LIN {X 0,Y 331.021,Z 915.228,A -85,B 0,C 180,E1 16163.029,E2 16163.029} C_VEL
LIN {X 0,Y 337.133,Z 895.779,A -85,B 0,C 180,E1 16164.723,E2 16164.723} C_VEL
LIN {X 0,Y 338.679,Z 881.099,A -85,B 0,C 180,E1 16166.333,E2 16166.333} C_VEL
LIN {X 0,Y 339.674,Z 868.031,A -85,B 0,C 180,E1 16167.682,E2 16167.682} C_VEL
LIN {X 0,Y 340.17,Z 866.046,A -85,B 0,C 180,E1 16167.812,E2 16167.812} C_VEL
LIN {X 0,Y 341.218,Z 861.378,A -85,B 0,C 180,E1 16168.096,E2 16168.096} C_VEL
LIN {X 0,Y 333.256,Z 836.302,A -85,B 0,C 180,E1 16172.609,E2 16172.609} C_VEL
LIN {X 0,Y 322.714,Z 812.784,A -85,B 0,C 180,E1 16178.041,E2 16178.041} C_VEL
LIN {X 0,Y 312.358,Z 794.085,A -85,B 0,C 180,E1 16183.992,E2 16183.992} C_VEL
LIN {X 0,Y 304.44,Z 781.718,A -85,B 0,C 180,E1 16189.789,E2 16189.789} C_VEL
LIN {X 0,Y 300.25,Z 775.211,A -85,B 0,C 180,E1 16194.023,E2 16194.023} C_VEL
LIN {X 0,Y 297.058,Z 768.999,A -85,B 0,C 180,E1 16199.536,E2 16199.536} C_VEL
LIN {X 0,Y 296.553,Z 769.306,A -85,B 0,C 180,E1 16209.301,E2 16209.301} C_VEL
LIN {X 0,Y 299.386,Z 775.096,A -85,B 0,C 180,E1 16215.012,E2 16215.012} C_VEL
LIN {X 0,Y 301.02,Z 777.25,A -85,B 0,C 180,E1 16217.046,E2 16217.046} C_VEL
LIN {X 0,Y 305.693,Z 785.45,A -85,B 0,C 180,E1 16221.795,E2 16221.795} C_VEL
LIN {X 0,Y 311.815,Z 796.017,A -85,B 0,C 180,E1 16226.634,E2 16226.634} C_VEL
LIN {X 0,Y 320.081,Z 813.536,A -85,B 0,C 180,E1 16232.477,E2 16232.477} C_VEL
LIN {X 0,Y 327.738,Z 835.588,A -85,B 0,C 180,E1 16238.25,E2 16238.25} C_VEL
LIN {X 0,Y 332.514,Z 859.666,A -85,B 0,C 180,E1 16243.601,E2 16243.601} C_VEL
LIN {X 0,Y 330.699,Z 866.985,A -85,B 0,C 180,E1 16244.544,E2 16244.544} C_VEL
LIN {X 0,Y 318.48,Z 897.247,A -85,B 0,C 180,E1 16248.528,E2 16248.528} C_VEL
LIN {X 0,Y 305.736,Z 923.66,A -85,B 0,C 180,E1 16253.542,E2 16253.542} C_VEL
LIN {X 0,Y 294.077,Z 945.097,A -85,B 0,C 180,E1 16259.443,E2 16259.443} C_VEL
LIN {X 0,Y 284.318,Z 962.198,A -85,B 0,C 180,E1 16266.461,E2 16266.461} C_VEL
LIN {X 0,Y 277.725,Z 974.062,A -85,B 0,C 180,E1 16274.183,E2 16274.183} C_VEL
LIN {X 0,Y 274.803,Z 979.693,A -85,B 0,C 180,E1 16280.487,E2 16280.487} C_VEL
LIN {X 0,Y 273.739,Z 982.416,A -85,B 0,C 180,E1 16286.83,E2 16286.83} C_VEL
LIN {X 0,Y 273.747,Z 982.384,A -85,B 0,C 180,E1 16293.171,E2 16293.171} C_VEL
LIN {X 0,Y 275.395,Z 978.493,A -85,B 0,C 180,E1 16301.094,E2 16301.094} C_VEL
LIN {X 0,Y 279.926,Z 969.8,A -85,B 0,C 180,E1 16308.936,E2 16308.936} C_VEL
LIN {X 0,Y 287.816,Z 955.85,A -85,B 0,C 180,E1 16316.395,E2 16316.395} C_VEL
LIN {X 0,Y 298.558,Z 936.897,A -85,B 0,C 180,E1 16322.978,E2 16322.978} C_VEL
LIN {X 0,Y 310.721,Z 913.541,A -85,B 0,C 180,E1 16328.506,E2 16328.506} C_VEL
LIN {X 0,Y 323.773,Z 884.724,A -85,B 0,C 180,E1 16333.206,E2 16333.206} C_VEL
LIN {X 0,Y 332.594,Z 860.778,A -85,B 0,C 180,E1 16336.051,E2 16336.051} C_VEL
LIN {X 0,Y 327.799,Z 836.283,A -85,B 0,C 180,E1 16341.479,E2 16341.479} C_VEL
LIN {X 0,Y 320.691,Z 815.062,A -85,B 0,C 180,E1 16346.924,E2 16346.924} C_VEL
LIN {X 0,Y 311.788,Z 796.082,A -85,B 0,C 180,E1 16353.185,E2 16353.185} C_VEL
LIN {X 0,Y 304.22,Z 782.321,A -85,B 0,C 180,E1 16359.432,E2 16359.432} C_VEL
LIN {X 0,Y 300.038,Z 775.489,A -85,B 0,C 180,E1 16363.895,E2 16363.895} C_VEL
LIN {X 0,Y 296.56,Z 769.453,A -85,B 0,C 180,E1 16369.925,E2 16369.925} C_VEL
LIN {X 0,Y 296.669,Z 768.461,A -85,B 0,C 180,E1 16380.008,E2 16380.008} C_VEL
LIN {X 0,Y 300.732,Z 775.566,A -85,B 0,C 180,E1 16386.693,E2 16386.693} C_VEL
LIN {X 0,Y 306.504,Z 785.112,A -85,B 0,C 180,E1 16392.034,E2 16392.034} C_VEL
LIN {X 0,Y 313.542,Z 796.189,A -85,B 0,C 180,E1 16396.847,E2 16396.847} C_VEL
LIN {X 0,Y 324.459,Z 816.254,A -85,B 0,C 180,E1 16402.919,E2 16402.919} C_VEL
LIN {X 0,Y 334.954,Z 840.847,A -85,B 0,C 180,E1 16408.338,E2 16408.338} C_VEL
LIN {X 0,Y 341.11,Z 861.37,A -85,B 0,C 180,E1 16411.908,E2 16411.908} C_VEL
LIN {X 0,Y 329.462,Z 902.909,A -85,B 0,C 180,E1 16414.862,E2 16414.862} C_VEL
LIN {X 0,Y 315.546,Z 942.717,A -85,B 0,C 180,E1 16419.055,E2 16419.055} C_VEL
LIN {X 0,Y 302.271,Z 976.846,A -85,B 0,C 180,E1 16424.232,E2 16424.232} C_VEL
LIN {X 0,Y 290.023,Z 1007.512,A -85,B 0,C 180,E1 16430.731,E2 16430.731} C_VEL
LIN {X 0,Y 280.658,Z 1033.018,A -85,B 0,C 180,E1 16438.227,E2 16438.227} C_VEL
LIN {X 0,Y 274.674,Z 1053.485,A -85,B 0,C 180,E1 16446.65,E2 16446.65} C_VEL
LIN {X 0,Y 272.304,Z 1067.457,A -85,B 0,C 180,E1 16455.096,E2 16455.096} C_VEL
LIN {X 0,Y 271.923,Z 1074.33,A -85,B 0,C 180,E1 16461.999,E2 16461.999} C_VEL
LIN {X 0,Y 272.108,Z 1076.824,A -85,B 0,C 180,E1 16466.81,E2 16466.81} C_VEL
LIN {X 0,Y 272.364,Z 1077.339,A -85,B 0,C 180,E1 16470,E2 16470} C_VEL
LIN {X 0,Y 272.002,Z 1075.42,A -85,B 0,C 180,E1 16476.391,E2 16476.391} C_VEL
LIN {X 0,Y 272.256,Z 1067.956,A -85,B 0,C 180,E1 16484.492,E2 16484.492} C_VEL
LIN {X 0,Y 274.36,Z 1054.719,A -85,B 0,C 180,E1 16492.723,E2 16492.723} C_VEL
LIN {X 0,Y 279.536,Z 1036.37,A -85,B 0,C 180,E1 16500.582,E2 16500.582} C_VEL
LIN {X 0,Y 288.648,Z 1011.145,A -85,B 0,C 180,E1 16508.341,E2 16508.341} C_VEL
LIN {X 0,Y 300.414,Z 981.675,A -85,B 0,C 180,E1 16514.874,E2 16514.874} C_VEL
LIN {X 0,Y 313.155,Z 949.302,A -85,B 0,C 180,E1 16520.072,E2 16520.072} C_VEL
LIN {X 0,Y 326.1,Z 913.314,A -85,B 0,C 180,E1 16524.199,E2 16524.199} C_VEL
LIN {X 0,Y 338.026,Z 873.973,A -85,B 0,C 180,E1 16527.32,E2 16527.32} C_VEL
LIN {X 0,Y 340.17,Z 866.046,A -85,B 0,C 180,E1 16527.812,E2 16527.812} C_VEL
LIN {X 0,Y 339.446,Z 860.887,A -85,B 0,C 180,E1 16528.559,E2 16528.559} C_VEL
LIN {X 0,Y 332.595,Z 853.241,A -85,B 0,C 180,E1 16530.955,E2 16530.955} C_VEL
LIN {X 0,Y 323.201,Z 827.838,A -85,B 0,C 180,E1 16536.348,E2 16536.348} C_VEL
LIN {X 0,Y 313.242,Z 807.134,A -85,B 0,C 180,E1 16542.23,E2 16542.23} C_VEL
LIN {X 0,Y 305.313,Z 793.908,A -85,B 0,C 180,E1 16547.736,E2 16547.736} C_VEL
LIN {X 0,Y 301.561,Z 787.929,A -85,B 0,C 180,E1 16551.058,E2 16551.058} C_VEL
LIN {X 0,Y 298.756,Z 782.824,A -85,B 0,C 180,E1 16554.358,E2 16554.358} C_VEL
LIN {X 0,Y 295.744,Z 776.422,A -85,B 0,C 180,E1 16559.992,E2 16559.992} C_VEL
LIN {X 0,Y 295.279,Z 777.204,A -85,B 0,C 180,E1 16569.164,E2 16569.164} C_VEL
LIN {X 0,Y 298.129,Z 783.012,A -85,B 0,C 180,E1 16575.301,E2 16575.301} C_VEL
LIN {X 0,Y 302.957,Z 791.913,A -85,B 0,C 180,E1 16581.04,E2 16581.04} C_VEL
LIN {X 0,Y 308.902,Z 803.163,A -85,B 0,C 180,E1 16586.27,E2 16586.27} C_VEL
LIN {X 0,Y 316.328,Z 820.365,A -85,B 0,C 180,E1 16592.16,E2 16592.16} C_VEL
LIN {X 0,Y 322.984,Z 841.616,A -85,B 0,C 180,E1 16597.876,E2 16597.876} C_VEL
LIN {X 0,Y 326.886,Z 864.273,A -85,B 0,C 180,E1 16603.076,E2 16603.076} C_VEL
LIN {X 0,Y 314.014,Z 895.921,A -85,B 0,C 180,E1 16607.129,E2 16607.129} C_VEL
LIN {X 0,Y 300.859,Z 922.582,A -85,B 0,C 180,E1 16612.083,E2 16612.083} C_VEL
LIN {X 0,Y 289.103,Z 943.576,A -85,B 0,C 180,E1 16617.687,E2 16617.687} C_VEL
LIN {X 0,Y 278.977,Z 960.478,A -85,B 0,C 180,E1 16624.269,E2 16624.269} C_VEL
LIN {X 0,Y 271.013,Z 973.81,A -85,B 0,C 180,E1 16632.406,E2 16632.406} C_VEL
LIN {X 0,Y 267.113,Z 981.045,A -85,B 0,C 180,E1 16640.21,E2 16640.21} C_VEL
LIN {X 0,Y 265.969,Z 983.764,A -85,B 0,C 180,E1 16646.737,E2 16646.737} C_VEL
LIN {X 0,Y 265.977,Z 983.732,A -85,B 0,C 180,E1 16653.263,E2 16653.263} C_VEL
LIN {X 0,Y 267.761,Z 979.844,A -85,B 0,C 180,E1 16661.414,E2 16661.414} C_VEL
LIN {X 0,Y 272.543,Z 971.167,A -85,B 0,C 180,E1 16669.47,E2 16669.47} C_VEL
LIN {X 0,Y 280.895,Z 957.141,A -85,B 0,C 180,E1 16677.143,E2 16677.143} C_VEL
LIN {X 0,Y 291.909,Z 938.548,A -85,B 0,C 180,E1 16683.739,E2 16683.739} C_VEL
LIN {X 0,Y 304.564,Z 915.214,A -85,B 0,C 180,E1 16689.374,E2 16689.374} C_VEL
LIN {X 0,Y 317.442,Z 887.919,A -85,B 0,C 180,E1 16693.931,E2 16693.931} C_VEL
LIN {X 0,Y 326.74,Z 863.857,A -85,B 0,C 180,E1 16696.906,E2 16696.906} C_VEL
LIN {X 0,Y 322.479,Z 840.057,A -85,B 0,C 180,E1 16702.399,E2 16702.399} C_VEL
LIN {X 0,Y 316.105,Z 820.038,A -85,B 0,C 180,E1 16707.814,E2 16707.814} C_VEL
LIN {X 0,Y 308.12,Z 801.577,A -85,B 0,C 180,E1 16714.168,E2 16714.168} C_VEL
LIN {X 0,Y 301.32,Z 789.044,A -85,B 0,C 180,E1 16720.375,E2 16720.375} C_VEL
LIN {X 0,Y 297.981,Z 782.896,A -85,B 0,C 180,E1 16724.538,E2 16724.538} C_VEL
LIN {X 0,Y 295.21,Z 776.702,A -85,B 0,C 180,E1 16730.495,E2 16730.495} C_VEL
LIN {X 0,Y 295.719,Z 776.954,A -85,B 0,C 180,E1 16740.649,E2 16740.649} C_VEL
LIN {X 0,Y 299.033,Z 783.061,A -85,B 0,C 180,E1 16746.183,E2 16746.183} C_VEL
LIN {X 0,Y 304.41,Z 792.508,A -85,B 0,C 180,E1 16751.663,E2 16751.663} C_VEL
LIN {X 0,Y 311.029,Z 803.407,A -85,B 0,C 180,E1 16756.442,E2 16756.442} C_VEL
LIN {X 0,Y 320.973,Z 822.87,A -85,B 0,C 180,E1 16762.449,E2 16762.449} C_VEL
LIN {X 0,Y 330.869,Z 847.763,A -85,B 0,C 180,E1 16768.028,E2 16768.028} C_VEL
LIN {X 0,Y 335.299,Z 865.581,A -85,B 0,C 180,E1 16771.117,E2 16771.117} C_VEL
LIN {X 0,Y 323.255,Z 905.592,A -85,B 0,C 180,E1 16774.067,E2 16774.067} C_VEL
LIN {X 0,Y 309.246,Z 943.627,A -85,B 0,C 180,E1 16778.197,E2 16778.197} C_VEL
LIN {X 0,Y 295.249,Z 977.945,A -85,B 0,C 180,E1 16783.568,E2 16783.568} C_VEL
LIN {X 0,Y 282.871,Z 1007.45,A -85,B 0,C 180,E1 16790.039,E2 16790.039} C_VEL
LIN {X 0,Y 273.077,Z 1032.74,A -85,B 0,C 180,E1 16797.749,E2 16797.749} C_VEL
LIN {X 0,Y 267.231,Z 1051.564,A -85,B 0,C 180,E1 16805.703,E2 16805.703} C_VEL
LIN {X 0,Y 264.59,Z 1065.504,A -85,B 0,C 180,E1 16814.229,E2 16814.229} C_VEL
LIN {X 0,Y 264.096,Z 1072.957,A -85,B 0,C 180,E1 16821.76,E2 16821.76} C_VEL
LIN {X 0,Y 264.307,Z 1075.47,A -85,B 0,C 180,E1 16826.716,E2 16826.716} C_VEL
LIN {X 0,Y 264.598,Z 1075.994,A -85,B 0,C 180,E1 16830,E2 16830} C_VEL
LIN {X 0,Y 264.197,Z 1074.056,A -85,B 0,C 180,E1 16836.581,E2 16836.581} C_VEL
LIN {X 0,Y 264.316,Z 1068.494,A -85,B 0,C 180,E1 16843.245,E2 16843.245} C_VEL
LIN {X 0,Y 266.059,Z 1056.461,A -85,B 0,C 180,E1 16851.708,E2 16851.708} C_VEL
LIN {X 0,Y 271.419,Z 1037.536,A -85,B 0,C 180,E1 16860.495,E2 16860.495} C_VEL
LIN {X 0,Y 280.433,Z 1013.604,A -85,B 0,C 180,E1 16868.343,E2 16868.343} C_VEL
LIN {X 0,Y 292.855,Z 983.925,A -85,B 0,C 180,E1 16875.303,E2 16875.303} C_VEL
LIN {X 0,Y 306.741,Z 950.365,A -85,B 0,C 180,E1 16880.896,E2 16880.896} C_VEL
LIN {X 0,Y 320.69,Z 913.175,A -85,B 0,C 180,E1 16885.243,E2 16885.243} C_VEL
LIN {X 0,Y 332.946,Z 874.288,A -85,B 0,C 180,E1 16888.358,E2 16888.358} C_VEL
LIN {X 0,Y 335.623,Z 864.362,A -85,B 0,C 180,E1 16888.991,E2 16888.991} C_VEL
LIN {X 0,Y 332.595,Z 853.241,A -85,B 0,C 180,E1 16890.955,E2 16890.955} C_VEL
LIN {X 0,Y 328.462,Z 846.564,A -85,B 0,C 180,E1 16892.778,E2 16892.778} C_VEL
LIN {X 0,Y 320.655,Z 837.361,A -85,B 0,C 180,E1 16896.065,E2 16896.065} C_VEL
LIN {X 0,Y 311.653,Z 817.013,A -85,B 0,C 180,E1 16901.77,E2 16901.77} C_VEL
LIN {X 0,Y 304.174,Z 802.822,A -85,B 0,C 180,E1 16907.233,E2 16907.233} C_VEL
LIN {X 0,Y 299.303,Z 794.888,A -85,B 0,C 180,E1 16911.722,E2 16911.722} C_VEL
LIN {X 0,Y 296.792,Z 790.23,A -85,B 0,C 180,E1 16914.871,E2 16914.871} C_VEL
LIN {X 0,Y 294.14,Z 784.145,A -85,B 0,C 180,E1 16920.61,E2 16920.61} C_VEL
LIN {X 0,Y 293.722,Z 784.97,A -85,B 0,C 180,E1 16928.968,E2 16928.968} C_VEL
LIN {X 0,Y 296.55,Z 790.82,A -85,B 0,C 180,E1 16935.482,E2 16935.482} C_VEL
LIN {X 0,Y 301.16,Z 800.76,A -85,B 0,C 180,E1 16941.462,E2 16941.462} C_VEL
LIN {X 0,Y 306.312,Z 811.538,A -85,B 0,C 180,E1 16946.402,E2 16946.402} C_VEL
LIN {X 0,Y 312.882,Z 828.141,A -85,B 0,C 180,E1 16952.148,E2 16952.148} C_VEL
LIN {X 0,Y 318.462,Z 848.77,A -85,B 0,C 180,E1 16957.799,E2 16957.799} C_VEL
LIN {X 0,Y 320.811,Z 868.378,A -85,B 0,C 180,E1 16962.364,E2 16962.364} C_VEL
LIN {X 0,Y 308.216,Z 897.773,A -85,B 0,C 180,E1 16966.206,E2 16966.206} C_VEL
LIN {X 0,Y 294.886,Z 923.817,A -85,B 0,C 180,E1 16971.112,E2 16971.112} C_VEL
LIN {X 0,Y 282.334,Z 945.309,A -85,B 0,C 180,E1 16976.958,E2 16976.958} C_VEL
LIN {X 0,Y 271.966,Z 961.846,A -85,B 0,C 180,E1 16983.555,E2 16983.555} C_VEL
LIN {X 0,Y 264.131,Z 974.24,A -85,B 0,C 180,E1 16991.125,E2 16991.125} C_VEL
LIN {X 0,Y 259.45,Z 982.392,A -85,B 0,C 180,E1 16999.918,E2 16999.918} C_VEL
LIN {X 0,Y 258.208,Z 985.111,A -85,B 0,C 180,E1 17006.639,E2 17006.639} C_VEL
LIN {X 0,Y 258.217,Z 985.079,A -85,B 0,C 180,E1 17013.362,E2 17013.362} C_VEL
LIN {X 0,Y 260.137,Z 981.196,A -85,B 0,C 180,E1 17021.754,E2 17021.754} C_VEL
LIN {X 0,Y 265.186,Z 972.532,A -85,B 0,C 180,E1 17030.033,E2 17030.033} C_VEL
LIN {X 0,Y 273.959,Z 958.549,A -85,B 0,C 180,E1 17037.872,E2 17037.872} C_VEL
LIN {X 0,Y 285.458,Z 939.958,A -85,B 0,C 180,E1 17044.608,E2 17044.608} C_VEL
LIN {X 0,Y 298.643,Z 916.602,A -85,B 0,C 180,E1 17050.333,E2 17050.333} C_VEL
LIN {X 0,Y 312.136,Z 888.985,A -85,B 0,C 180,E1 17054.985,E2 17054.985} C_VEL
LIN {X 0,Y 320.922,Z 866.987,A -85,B 0,C 180,E1 17057.772,E2 17057.772} C_VEL
LIN {X 0,Y 317.398,Z 844.495,A -85,B 0,C 180,E1 17063.182,E2 17063.182} C_VEL
LIN {X 0,Y 311.442,Z 824.288,A -85,B 0,C 180,E1 17068.913,E2 17068.913} C_VEL
LIN {X 0,Y 304.534,Z 807.578,A -85,B 0,C 180,E1 17075.06,E2 17075.06} C_VEL
LIN {X 0,Y 298.817,Z 796.122,A -85,B 0,C 180,E1 17080.974,E2 17080.974} C_VEL
LIN {X 0,Y 296.046,Z 790.466,A -85,B 0,C 180,E1 17084.815,E2 17084.815} C_VEL
LIN {X 0,Y 293.489,Z 784.102,A -85,B 0,C 180,E1 17091.354,E2 17091.354} C_VEL
LIN {X 0,Y 294.251,Z 784.854,A -85,B 0,C 180,E1 17100.484,E2 17100.484} C_VEL
LIN {X 0,Y 298.156,Z 792.625,A -85,B 0,C 180,E1 17107.117,E2 17107.117} C_VEL
LIN {X 0,Y 303.043,Z 801.272,A -85,B 0,C 180,E1 17111.991,E2 17111.991} C_VEL
LIN {X 0,Y 310.547,Z 814.766,A -85,B 0,C 180,E1 17117.563,E2 17117.563} C_VEL
LIN {X 0,Y 319.314,Z 834.216,A -85,B 0,C 180,E1 17123.176,E2 17123.176} C_VEL
LIN {X 0,Y 327.303,Z 857.161,A -85,B 0,C 180,E1 17128.233,E2 17128.233} C_VEL
LIN {X 0,Y 329.873,Z 867.279,A -85,B 0,C 180,E1 17130.105,E2 17130.105} C_VEL
LIN {X 0,Y 317.632,Z 906.603,A -85,B 0,C 180,E1 17133.096,E2 17133.096} C_VEL
LIN {X 0,Y 303.691,Z 942.962,A -85,B 0,C 180,E1 17137.094,E2 17137.094} C_VEL
LIN {X 0,Y 289.455,Z 976.399,A -85,B 0,C 180,E1 17142.37,E2 17142.37} C_VEL
LIN {X 0,Y 276.484,Z 1005.907,A -85,B 0,C 180,E1 17148.92,E2 17148.92} C_VEL
LIN {X 0,Y 265.97,Z 1031.227,A -85,B 0,C 180,E1 17156.778,E2 17156.778} C_VEL
LIN {X 0,Y 259.706,Z 1050.107,A -85,B 0,C 180,E1 17164.951,E2 17164.951} C_VEL
LIN {X 0,Y 256.828,Z 1064.091,A -85,B 0,C 180,E1 17173.739,E2 17173.739} C_VEL
LIN {X 0,Y 256.281,Z 1071.587,A -85,B 0,C 180,E1 17181.507,E2 17181.507} C_VEL
LIN {X 0,Y 256.513,Z 1074.116,A -85,B 0,C 180,E1 17186.616,E2 17186.616} C_VEL
LIN {X 0,Y 256.824,Z 1074.647,A -85,B 0,C 180,E1 17190,E2 17190} C_VEL
LIN {X 0,Y 256.363,Z 1072.688,A -85,B 0,C 180,E1 17196.783,E2 17196.783} C_VEL
LIN {X 0,Y 256.514,Z 1067.096,A -85,B 0,C 180,E1 17203.655,E2 17203.655} C_VEL
LIN {X 0,Y 258.399,Z 1055.007,A -85,B 0,C 180,E1 17212.386,E2 17212.386} C_VEL
LIN {X 0,Y 264.325,Z 1035.788,A -85,B 0,C 180,E1 17221.51,E2 17221.51} C_VEL
LIN {X 0,Y 274.32,Z 1010.866,A -85,B 0,C 180,E1 17229.767,E2 17229.767} C_VEL
LIN {X 0,Y 287.754,Z 980.553,A -85,B 0,C 180,E1 17236.838,E2 17236.838} C_VEL
LIN {X 0,Y 301.735,Z 948.101,A -85,B 0,C 180,E1 17242.211,E2 17242.211} C_VEL
LIN {X 0,Y 315.862,Z 911.832,A -85,B 0,C 180,E1 17246.427,E2 17246.427} C_VEL
LIN {X 0,Y 328.463,Z 872.948,A -85,B 0,C 180,E1 17249.529,E2 17249.529} C_VEL
LIN {X 0,Y 329.734,Z 866.231,A -85,B 0,C 180,E1 17250.095,E2 17250.095} C_VEL
LIN {X 0,Y 322.374,Z 841.982,A -85,B 0,C 180,E1 17254.991,E2 17254.991} C_VEL
LIN {X 0,Y 320.655,Z 837.361,A -85,B 0,C 180,E1 17256.065,E2 17256.065} C_VEL
LIN {X 0,Y 315.045,Z 830.532,A -85,B 0,C 180,E1 17258.785,E2 17258.785} C_VEL
LIN {X 0,Y 309.157,Z 825.25,A -85,B 0,C 180,E1 17261.716,E2 17261.716} C_VEL
LIN {X 0,Y 301.715,Z 810.065,A -85,B 0,C 180,E1 17267.588,E2 17267.588} C_VEL
LIN {X 0,Y 295.456,Z 798.281,A -85,B 0,C 180,E1 17274.486,E2 17274.486} C_VEL
LIN {X 0,Y 292.411,Z 791.833,A -85,B 0,C 180,E1 17281.236,E2 17281.236} C_VEL
LIN {X 0,Y 292.006,Z 792.598,A -85,B 0,C 180,E1 17288.705,E2 17288.705} C_VEL
LIN {X 0,Y 294.956,Z 799.949,A -85,B 0,C 180,E1 17296.197,E2 17296.197} C_VEL
LIN {X 0,Y 299.591,Z 809.865,A -85,B 0,C 180,E1 17302.264,E2 17302.264} C_VEL
LIN {X 0,Y 306.256,Z 826.745,A -85,B 0,C 180,E1 17309.179,E2 17309.179} C_VEL
LIN {X 0,Y 311.878,Z 846.274,A -85,B 0,C 180,E1 17315.19,E2 17315.19} C_VEL
LIN {X 0,Y 315.042,Z 867.402,A -85,B 0,C 180,E1 17320.56,E2 17320.56} C_VEL
LIN {X 0,Y 314.79,Z 872.158,A -85,B 0,C 180,E1 17321.568,E2 17321.568} C_VEL
LIN {X 0,Y 301.976,Z 900.685,A -85,B 0,C 180,E1 17325.42,E2 17325.42} C_VEL
LIN {X 0,Y 287.935,Z 926.863,A -85,B 0,C 180,E1 17330.519,E2 17330.519} C_VEL
LIN {X 0,Y 274.877,Z 948.177,A -85,B 0,C 180,E1 17336.579,E2 17336.579} C_VEL
LIN {X 0,Y 263.958,Z 964.767,A -85,B 0,C 180,E1 17343.608,E2 17343.608} C_VEL
LIN {X 0,Y 256.205,Z 976.415,A -85,B 0,C 180,E1 17351.25,E2 17351.25} C_VEL
LIN {X 0,Y 251.774,Z 983.743,A -85,B 0,C 180,E1 17359.607,E2 17359.607} C_VEL
LIN {X 0,Y 250.439,Z 986.459,A -85,B 0,C 180,E1 17366.534,E2 17366.534} C_VEL
LIN {X 0,Y 250.449,Z 986.427,A -85,B 0,C 180,E1 17373.466,E2 17373.466} C_VEL
LIN {X 0,Y 252.502,Z 982.55,A -85,B 0,C 180,E1 17382.114,E2 17382.114} C_VEL
LIN {X 0,Y 257.855,Z 973.896,A -85,B 0,C 180,E1 17390.628,E2 17390.628} C_VEL
LIN {X 0,Y 267.09,Z 959.928,A -85,B 0,C 180,E1 17398.654,E2 17398.654} C_VEL
LIN {X 0,Y 279.246,Z 941.078,A -85,B 0,C 180,E1 17405.605,E2 17405.605} C_VEL
LIN {X 0,Y 292.765,Z 918.055,A -85,B 0,C 180,E1 17411.317,E2 17411.317} C_VEL
LIN {X 0,Y 307.165,Z 889.619,A -85,B 0,C 180,E1 17416.131,E2 17416.131} C_VEL
LIN {X 0,Y 315.16,Z 870.376,A -85,B 0,C 180,E1 17418.59,E2 17418.59} C_VEL
LIN {X 0,Y 312.312,Z 849.014,A -85,B 0,C 180,E1 17423.972,E2 17423.972} C_VEL
LIN {X 0,Y 307.176,Z 829.742,A -85,B 0,C 180,E1 17429.667,E2 17429.667} C_VEL
LIN {X 0,Y 301.322,Z 814.349,A -85,B 0,C 180,E1 17435.52,E2 17435.52} C_VEL
LIN {X 0,Y 296.413,Z 803.533,A -85,B 0,C 180,E1 17441.2,E2 17441.2} C_VEL
LIN {X 0,Y 293.878,Z 797.833,A -85,B 0,C 180,E1 17445.273,E2 17445.273} C_VEL
LIN {X 0,Y 291.776,Z 791.801,A -85,B 0,C 180,E1 17451.773,E2 17451.773} C_VEL
LIN {X 0,Y 292.61,Z 792.48,A -85,B 0,C 180,E1 17460.168,E2 17460.168} C_VEL
LIN {X 0,Y 296.269,Z 800.424,A -85,B 0,C 180,E1 17466.982,E2 17466.982} C_VEL
LIN {X 0,Y 302.189,Z 810.993,A -85,B 0,C 180,E1 17472.944,E2 17472.944} C_VEL
LIN {X 0,Y 310.622,Z 828.689,A -85,B 0,C 180,E1 17479.397,E2 17479.397} C_VEL
LIN {X 0,Y 318.81,Z 850.034,A -85,B 0,C 180,E1 17485.005,E2 17485.005} C_VEL
LIN {X 0,Y 324.236,Z 870.946,A -85,B 0,C 180,E1 17489.244,E2 17489.244} C_VEL
LIN {X 0,Y 311.88,Z 908.2,A -85,B 0,C 180,E1 17492.142,E2 17492.142} C_VEL
LIN {X 0,Y 297.637,Z 943.741,A -85,B 0,C 180,E1 17496.146,E2 17496.146} C_VEL
LIN {X 0,Y 282.903,Z 976.713,A -85,B 0,C 180,E1 17501.476,E2 17501.476} C_VEL
LIN {X 0,Y 269.332,Z 1006.106,A -85,B 0,C 180,E1 17508.215,E2 17508.215} C_VEL
LIN {X 0,Y 258.453,Z 1030.924,A -85,B 0,C 180,E1 17516.219,E2 17516.219} C_VEL
LIN {X 0,Y 251.677,Z 1050.333,A -85,B 0,C 180,E1 17525.096,E2 17525.096} C_VEL
LIN {X 0,Y 248.898,Z 1063.731,A -85,B 0,C 180,E1 17534.114,E2 17534.114} C_VEL
LIN {X 0,Y 248.452,Z 1070.213,A -85,B 0,C 180,E1 17541.237,E2 17541.237} C_VEL
LIN {X 0,Y 248.708,Z 1072.761,A -85,B 0,C 180,E1 17546.51,E2 17546.51} C_VEL
LIN {X 0,Y 249.056,Z 1073.302,A -85,B 0,C 180,E1 17550,E2 17550} C_VEL
LIN {X 0,Y 248.529,Z 1071.319,A -85,B 0,C 180,E1 17556.998,E2 17556.998} C_VEL
LIN {X 0,Y 248.715,Z 1065.697,A -85,B 0,C 180,E1 17564.092,E2 17564.092} C_VEL
LIN {X 0,Y 250.807,Z 1053.558,A -85,B 0,C 180,E1 17573.102,E2 17573.102} C_VEL
LIN {X 0,Y 257.19,Z 1034.307,A -85,B 0,C 180,E1 17582.481,E2 17582.481} C_VEL
LIN {X 0,Y 267.66,Z 1009.741,A -85,B 0,C 180,E1 17590.811,E2 17590.811} C_VEL
LIN {X 0,Y 281.601,Z 979.841,A -85,B 0,C 180,E1 17597.921,E2 17597.921} C_VEL
LIN {X 0,Y 296.65,Z 946.39,A -85,B 0,C 180,E1 17603.496,E2 17603.496} C_VEL
LIN {X 0,Y 311.043,Z 910.806,A -85,B 0,C 180,E1 17607.622,E2 17607.622} C_VEL
LIN {X 0,Y 324.005,Z 872.104,A -85,B 0,C 180,E1 17610.694,E2 17610.694} C_VEL
LIN {X 0,Y 323.385,Z 866.163,A -85,B 0,C 180,E1 17611.649,E2 17611.649} C_VEL
LIN {X 0,Y 316.564,Z 843.36,A -85,B 0,C 180,E1 17616.615,E2 17616.615} C_VEL
LIN {X 0,Y 309.157,Z 825.25,A -85,B 0,C 180,E1 17621.716,E2 17621.716} C_VEL
LIN {X 0,Y 303.851,Z 820.892,A -85,B 0,C 180,E1 17624.739,E2 17624.739} C_VEL
LIN {X 0,Y 299.105,Z 817.316,A -85,B 0,C 180,E1 17627.905,E2 17627.905} C_VEL
LIN {X 0,Y 293.296,Z 805.737,A -85,B 0,C 180,E1 17634.824,E2 17634.824} C_VEL
LIN {X 0,Y 290.6,Z 799.522,A -85,B 0,C 180,E1 17641.243,E2 17641.243} C_VEL
LIN {X 0,Y 290.119,Z 800.333,A -85,B 0,C 180,E1 17648.577,E2 17648.577} C_VEL
LIN {X 0,Y 292.552,Z 807.429,A -85,B 0,C 180,E1 17655.948,E2 17655.948} C_VEL
LIN {X 0,Y 296.428,Z 816.63,A -85,B 0,C 180,E1 17661.724,E2 17661.724} C_VEL
LIN {X 0,Y 302.091,Z 832.275,A -85,B 0,C 180,E1 17668.421,E2 17668.421} C_VEL
LIN {X 0,Y 307.045,Z 851.682,A -85,B 0,C 180,E1 17674.621,E2 17674.621} C_VEL
LIN {X 0,Y 309.442,Z 872.145,A -85,B 0,C 180,E1 17680.028,E2 17680.028} C_VEL
LIN {X 0,Y 308.896,Z 875.778,A -85,B 0,C 180,E1 17680.724,E2 17680.724} C_VEL
LIN {X 0,Y 294.572,Z 906.129,A -85,B 0,C 180,E1 17685.033,E2 17685.033} C_VEL
LIN {X 0,Y 279.552,Z 932.288,A -85,B 0,C 180,E1 17690.48,E2 17690.48} C_VEL
LIN {X 0,Y 265.599,Z 953.756,A -85,B 0,C 180,E1 17697.213,E2 17697.213} C_VEL
LIN {X 0,Y 254.953,Z 969.085,A -85,B 0,C 180,E1 17704.499,E2 17704.499} C_VEL
LIN {X 0,Y 247.761,Z 979.488,A -85,B 0,C 180,E1 17712.21,E2 17712.21} C_VEL
LIN {X 0,Y 244.128,Z 985.091,A -85,B 0,C 180,E1 17719.278,E2 17719.278} C_VEL
LIN {X 0,Y 242.674,Z 987.807,A -85,B 0,C 180,E1 17726.423,E2 17726.423} C_VEL
LIN {X 0,Y 242.701,Z 987.731,A -85,B 0,C 180,E1 17733.758,E2 17733.758} C_VEL
LIN {X 0,Y 245.737,Z 982.562,A -85,B 0,C 180,E1 17744.267,E2 17744.267} C_VEL
LIN {X 0,Y 253.133,Z 971.629,A -85,B 0,C 180,E1 17753.811,E2 17753.811} C_VEL
LIN {X 0,Y 264.331,Z 955.472,A -85,B 0,C 180,E1 17761.993,E2 17761.993} C_VEL
LIN {X 0,Y 277.967,Z 934.637,A -85,B 0,C 180,E1 17768.783,E2 17768.783} C_VEL
LIN {X 0,Y 292.633,Z 909.354,A -85,B 0,C 180,E1 17774.303,E2 17774.303} C_VEL
LIN {X 0,Y 307.302,Z 879.317,A -85,B 0,C 180,E1 17778.741,E2 17778.741} C_VEL
LIN {X 0,Y 309.41,Z 873.088,A -85,B 0,C 180,E1 17779.614,E2 17779.614} C_VEL
LIN {X 0,Y 306.805,Z 851.1,A -85,B 0,C 180,E1 17785.438,E2 17785.438} C_VEL
LIN {X 0,Y 301.882,Z 831.98,A -85,B 0,C 180,E1 17791.558,E2 17791.558} C_VEL
LIN {X 0,Y 296.201,Z 816.357,A -85,B 0,C 180,E1 17798.258,E2 17798.258} C_VEL
LIN {X 0,Y 291.569,Z 805.297,A -85,B 0,C 180,E1 17805.538,E2 17805.538} C_VEL
LIN {X 0,Y 289.948,Z 799.47,A -85,B 0,C 180,E1 17811.753,E2 17811.753} C_VEL
LIN {X 0,Y 290.704,Z 800.229,A -85,B 0,C 180,E1 17820.008,E2 17820.008} C_VEL
LIN {X 0,Y 294.115,Z 807.974,A -85,B 0,C 180,E1 17826.729,E2 17826.729} C_VEL
LIN {X 0,Y 299.472,Z 818.255,A -85,B 0,C 180,E1 17832.599,E2 17832.599} C_VEL
LIN {X 0,Y 306.638,Z 834.37,A -85,B 0,C 180,E1 17838.629,E2 17838.629} C_VEL
LIN {X 0,Y 314.015,Z 854.697,A -85,B 0,C 180,E1 17844.198,E2 17844.198} C_VEL
LIN {X 0,Y 318.669,Z 872.859,A -85,B 0,C 180,E1 17848.106,E2 17848.106} C_VEL
LIN {X 0,Y 304.476,Z 914.383,A -85,B 0,C 180,E1 17851.601,E2 17851.601} C_VEL
LIN {X 0,Y 288.852,Z 950.821,A -85,B 0,C 180,E1 17856.054,E2 17856.054} C_VEL
LIN {X 0,Y 273.166,Z 983.833,A -85,B 0,C 180,E1 17861.941,E2 17861.941} C_VEL
LIN {X 0,Y 259.286,Z 1012.376,A -85,B 0,C 180,E1 17869.248,E2 17869.248} C_VEL
LIN {X 0,Y 248.714,Z 1036.11,A -85,B 0,C 180,E1 17877.925,E2 17877.925} C_VEL
LIN {X 0,Y 242.801,Z 1053.526,A -85,B 0,C 180,E1 17887.063,E2 17887.063} C_VEL
LIN {X 0,Y 240.929,Z 1064.285,A -85,B 0,C 180,E1 17895.442,E2 17895.442} C_VEL
LIN {X 0,Y 240.728,Z 1069.947,A -85,B 0,C 180,E1 17902.774,E2 17902.774} C_VEL
LIN {X 0,Y 241.272,Z 1071.953,A -85,B 0,C 180,E1 17910,E2 17910} C_VEL
LIN {X 0,Y 240.719,Z 1069.953,A -85,B 0,C 180,E1 17917.226,E2 17917.226} C_VEL
LIN {X 0,Y 240.917,Z 1064.297,A -85,B 0,C 180,E1 17924.558,E2 17924.558} C_VEL
LIN {X 0,Y 243.211,Z 1052.103,A -85,B 0,C 180,E1 17933.867,E2 17933.867} C_VEL
LIN {X 0,Y 250.08,Z 1032.856,A -85,B 0,C 180,E1 17943.498,E2 17943.498} C_VEL
LIN {X 0,Y 261.205,Z 1008.5,A -85,B 0,C 180,E1 17951.933,E2 17951.933} C_VEL
LIN {X 0,Y 275.677,Z 978.942,A -85,B 0,C 180,E1 17959.083,E2 17959.083} C_VEL
LIN {X 0,Y 291.044,Z 946.214,A -85,B 0,C 180,E1 17964.618,E2 17964.618} C_VEL
LIN {X 0,Y 306.252,Z 910.007,A -85,B 0,C 180,E1 17968.839,E2 17968.839} C_VEL
LIN {X 0,Y 318.781,Z 872.955,A -85,B 0,C 180,E1 17971.891,E2 17971.891} C_VEL
LIN {X 0,Y 312.641,Z 850.178,A -85,B 0,C 180,E1 17976.939,E2 17976.939} C_VEL
LIN {X 0,Y 304.74,Z 829.528,A -85,B 0,C 180,E1 17983.023,E2 17983.023} C_VEL
LIN {X 0,Y 299.105,Z 817.316,A -85,B 0,C 180,E1 17987.905,E2 17987.905} C_VEL
LIN {X 0,Y 295.74,Z 817.261,A -85,B 0,C 180,E1 17990.084,E2 17990.084} C_VEL
LIN {X 0,Y 292.707,Z 817.502,A -85,B 0,C 180,E1 17992.324,E2 17992.324} C_VEL
LIN {X 0,Y 290.344,Z 812.431,A -85,B 0,C 180,E1 17996.079,E2 17996.079} C_VEL
LIN {X 0,Y 288.685,Z 807.185,A -85,B 0,C 180,E1 18001.252,E2 18001.252} C_VEL
LIN {X 0,Y 287.984,Z 807.868,A -85,B 0,C 180,E1 18008.323,E2 18008.323} C_VEL
LIN {X 0,Y 290.038,Z 815.136,A -85,B 0,C 180,E1 18015.852,E2 18015.852} C_VEL
LIN {X 0,Y 293.631,Z 824.651,A -85,B 0,C 180,E1 18021.861,E2 18021.861} C_VEL
LIN {X 0,Y 298.583,Z 840.335,A -85,B 0,C 180,E1 18028.561,E2 18028.561} C_VEL
LIN {X 0,Y 302.406,Z 858.826,A -85,B 0,C 180,E1 18034.546,E2 18034.546} C_VEL
LIN {X 0,Y 303.862,Z 877.43,A -85,B 0,C 180,E1 18039.609,E2 18039.609} C_VEL
LIN {X 0,Y 289.142,Z 907.625,A -85,B 0,C 180,E1 18043.948,E2 18043.948} C_VEL
LIN {X 0,Y 273.604,Z 933.695,A -85,B 0,C 180,E1 18049.445,E2 18049.445} C_VEL
LIN {X 0,Y 259.069,Z 955.133,A -85,B 0,C 180,E1 18056.277,E2 18056.277} C_VEL
LIN {X 0,Y 247.914,Z 970.449,A -85,B 0,C 180,E1 18063.721,E2 18063.721} C_VEL
LIN {X 0,Y 240.332,Z 980.841,A -85,B 0,C 180,E1 18071.641,E2 18071.641} C_VEL
LIN {X 0,Y 236.467,Z 986.441,A -85,B 0,C 180,E1 18078.926,E2 18078.926} C_VEL
LIN {X 0,Y 234.899,Z 989.156,A -85,B 0,C 180,E1 18086.305,E2 18086.305} C_VEL
LIN {X 0,Y 234.926,Z 989.122,A -85,B 0,C 180,E1 18093.695,E2 18093.695} C_VEL
LIN {X 0,Y 237.285,Z 985.257,A -85,B 0,C 180,E1 18102.904,E2 18102.904} C_VEL
LIN {X 0,Y 243.29,Z 976.622,A -85,B 0,C 180,E1 18111.924,E2 18111.924} C_VEL
LIN {X 0,Y 253.556,Z 962.576,A -85,B 0,C 180,E1 18120.4,E2 18120.4} C_VEL
LIN {X 0,Y 266.636,Z 944.03,A -85,B 0,C 180,E1 18127.51,E2 18127.51} C_VEL
LIN {X 0,Y 281.815,Z 920.132,A -85,B 0,C 180,E1 18133.57,E2 18133.57} C_VEL
LIN {X 0,Y 296.563,Z 892.868,A -85,B 0,C 180,E1 18138.265,E2 18138.265} C_VEL
LIN {X 0,Y 303.779,Z 877.043,A -85,B 0,C 180,E1 18140.364,E2 18140.364} C_VEL
LIN {X 0,Y 301.928,Z 856.582,A -85,B 0,C 180,E1 18145.989,E2 18145.989} C_VEL
LIN {X 0,Y 297.816,Z 838.046,A -85,B 0,C 180,E1 18152.142,E2 18152.142} C_VEL
LIN {X 0,Y 292.983,Z 823.069,A -85,B 0,C 180,E1 18158.804,E2 18158.804} C_VEL
LIN {X 0,Y 289.661,Z 813.515,A -85,B 0,C 180,E1 18164.86,E2 18164.86} C_VEL
LIN {X 0,Y 287.847,Z 807.072,A -85,B 0,C 180,E1 18172.038,E2 18172.038} C_VEL
LIN {X 0,Y 288.697,Z 807.845,A -85,B 0,C 180,E1 18179.801,E2 18179.801} C_VEL
LIN {X 0,Y 291.698,Z 815.388,A -85,B 0,C 180,E1 18186.442,E2 18186.442} C_VEL
LIN {X 0,Y 296.688,Z 825.553,A -85,B 0,C 180,E1 18192.275,E2 18192.275} C_VEL
LIN {X 0,Y 303.843,Z 842.834,A -85,B 0,C 180,E1 18198.784,E2 18198.784} C_VEL
LIN {X 0,Y 310.453,Z 864.042,A -85,B 0,C 180,E1 18204.495,E2 18204.495} C_VEL
LIN {X 0,Y 313.122,Z 877.427,A -85,B 0,C 180,E1 18207.343,E2 18207.343} C_VEL
LIN {X 0,Y 298.904,Z 915.633,A -85,B 0,C 180,E1 18210.562,E2 18210.562} C_VEL
LIN {X 0,Y 283.226,Z 950.728,A -85,B 0,C 180,E1 18214.921,E2 18214.921} C_VEL
LIN {X 0,Y 267.278,Z 982.828,A -85,B 0,C 180,E1 18220.72,E2 18220.72} C_VEL
LIN {X 0,Y 252.496,Z 1011.602,A -85,B 0,C 180,E1 18228.231,E2 18228.231} C_VEL
LIN {X 0,Y 241.75,Z 1034.421,A -85,B 0,C 180,E1 18236.776,E2 18236.776} C_VEL
LIN {X 0,Y 235.201,Z 1052.166,A -85,B 0,C 180,E1 18246.336,E2 18246.336} C_VEL
LIN {X 0,Y 233.12,Z 1062.878,A -85,B 0,C 180,E1 18254.943,E2 18254.943} C_VEL
LIN {X 0,Y 232.887,Z 1068.575,A -85,B 0,C 180,E1 18262.529,E2 18262.529} C_VEL
LIN {X 0,Y 233.501,Z 1070.607,A -85,B 0,C 180,E1 18270,E2 18270} C_VEL
LIN {X 0,Y 232.879,Z 1068.582,A -85,B 0,C 180,E1 18277.471,E2 18277.471} C_VEL
LIN {X 0,Y 233.108,Z 1062.892,A -85,B 0,C 180,E1 18285.057,E2 18285.057} C_VEL
LIN {X 0,Y 235.6,Z 1050.869,A -85,B 0,C 180,E1 18294.55,E2 18294.55} C_VEL
LIN {X 0,Y 242.626,Z 1032.391,A -85,B 0,C 180,E1 18304.166,E2 18304.166} C_VEL
LIN {X 0,Y 254.825,Z 1007.317,A -85,B 0,C 180,E1 18313.098,E2 18313.098} C_VEL
LIN {X 0,Y 270.176,Z 977.324,A -85,B 0,C 180,E1 18320.449,E2 18320.449} C_VEL
LIN {X 0,Y 286.369,Z 944.271,A -85,B 0,C 180,E1 18326.024,E2 18326.024} C_VEL
LIN {X 0,Y 301.77,Z 908.824,A -85,B 0,C 180,E1 18330.127,E2 18330.127} C_VEL
LIN {X 0,Y 313.217,Z 876.007,A -85,B 0,C 180,E1 18332.902,E2 18332.902} C_VEL
LIN {X 0,Y 307.75,Z 854.314,A -85,B 0,C 180,E1 18337.963,E2 18337.963} C_VEL
LIN {X 0,Y 300.79,Z 834.931,A -85,B 0,C 180,E1 18343.922,E2 18343.922} C_VEL
LIN {X 0,Y 294.61,Z 821.309,A -85,B 0,C 180,E1 18350.023,E2 18350.023} C_VEL
LIN {X 0,Y 292.707,Z 817.502,A -85,B 0,C 180,E1 18352.324,E2 18352.324} C_VEL
LIN {X 0,Y 290.213,Z 816.654,A -85,B 0,C 180,E1 18354.857,E2 18354.857} C_VEL
LIN {X 0,Y 286.752,Z 817.222,A -85,B 0,C 180,E1 18359.196,E2 18359.196} C_VEL
LIN {X 0,Y 286.226,Z 814.658,A -85,B 0,C 180,E1 18362.143,E2 18362.143} C_VEL
LIN {X 0,Y 285.724,Z 814.639,A -85,B 0,C 180,E1 18366.075,E2 18366.075} C_VEL
LIN {X 0,Y 287.227,Z 821.941,A -85,B 0,C 180,E1 18375.272,E2 18375.272} C_VEL
LIN {X 0,Y 290.683,Z 832.844,A -85,B 0,C 180,E1 18382.094,E2 18382.094} C_VEL
LIN {X 0,Y 294.563,Z 847.501,A -85,B 0,C 180,E1 18388.433,E2 18388.433} C_VEL
LIN {X 0,Y 297.575,Z 865.896,A -85,B 0,C 180,E1 18394.507,E2 18394.507} C_VEL
LIN {X 0,Y 298.272,Z 880.517,A -85,B 0,C 180,E1 18398.613,E2 18398.613} C_VEL
LIN {X 0,Y 282.723,Z 910.925,A -85,B 0,C 180,E1 18403.146,E2 18403.146} C_VEL
LIN {X 0,Y 266.809,Z 936.457,A -85,B 0,C 180,E1 18408.727,E2 18408.727} C_VEL
LIN {X 0,Y 252.61,Z 956.512,A -85,B 0,C 180,E1 18415.294,E2 18415.294} C_VEL
LIN {X 0,Y 240.935,Z 971.808,A -85,B 0,C 180,E1 18422.898,E2 18422.898} C_VEL
LIN {X 0,Y 232.908,Z 982.198,A -85,B 0,C 180,E1 18431.034,E2 18431.034} C_VEL
LIN {X 0,Y 228.817,Z 987.793,A -85,B 0,C 180,E1 18438.551,E2 18438.551} C_VEL
LIN {X 0,Y 227.087,Z 990.749,A -85,B 0,C 180,E1 18448.834,E2 18448.834} C_VEL
LIN {X 0,Y 227.669,Z 989.45,A -85,B 0,C 180,E1 18457.643,E2 18457.643} C_VEL
LIN {X 0,Y 231.678,Z 983.749,A -85,B 0,C 180,E1 18467.102,E2 18467.102} C_VEL
LIN {X 0,Y 239.948,Z 972.993,A -85,B 0,C 180,E1 18476.211,E2 18476.211} C_VEL
LIN {X 0,Y 251.226,Z 958.242,A -85,B 0,C 180,E1 18483.879,E2 18483.879} C_VEL
LIN {X 0,Y 266.02,Z 937.464,A -85,B 0,C 180,E1 18490.882,E2 18490.882} C_VEL
LIN {X 0,Y 281.743,Z 912.302,A -85,B 0,C 180,E1 18496.506,E2 18496.506} C_VEL
LIN {X 0,Y 296.707,Z 883.796,A -85,B 0,C 180,E1 18500.816,E2 18500.816} C_VEL
LIN {X 0,Y 298.169,Z 879.453,A -85,B 0,C 180,E1 18501.55,E2 18501.55} C_VEL
LIN {X 0,Y 296.574,Z 858.655,A -85,B 0,C 180,E1 18507.599,E2 18507.599} C_VEL
LIN {X 0,Y 292.946,Z 841.125,A -85,B 0,C 180,E1 18513.928,E2 18513.928} C_VEL
LIN {X 0,Y 288.865,Z 827.575,A -85,B 0,C 180,E1 18520.633,E2 18520.633} C_VEL
LIN {X 0,Y 286.41,Z 820.001,A -85,B 0,C 180,E1 18526.252,E2 18526.252} C_VEL
LIN {X 0,Y 285.5,Z 815.679,A -85,B 0,C 180,E1 18531.336,E2 18531.336} C_VEL
LIN {X 0,Y 285.775,Z 814.509,A -85,B 0,C 180,E1 18536.971,E2 18536.971} C_VEL
LIN {X 0,Y 286.421,Z 815.71,A -85,B 0,C 180,E1 18539.8,E2 18539.8} C_VEL
LIN {X 0,Y 289.13,Z 822.516,A -85,B 0,C 180,E1 18546.019,E2 18546.019} C_VEL
LIN {X 0,Y 294.009,Z 833.67,A -85,B 0,C 180,E1 18552.389,E2 18552.389} C_VEL
LIN {X 0,Y 300.306,Z 850.382,A -85,B 0,C 180,E1 18558.663,E2 18558.663} C_VEL
LIN {X 0,Y 306.32,Z 871.816,A -85,B 0,C 180,E1 18564.458,E2 18564.458} C_VEL
LIN {X 0,Y 307.483,Z 880.916,A -85,B 0,C 180,E1 18566.365,E2 18566.365} C_VEL
LIN {X 0,Y 292.838,Z 918.282,A -85,B 0,C 180,E1 18569.632,E2 18569.632} C_VEL
LIN {X 0,Y 277.008,Z 952.015,A -85,B 0,C 180,E1 18573.952,E2 18573.952} C_VEL
LIN {X 0,Y 260.972,Z 982.807,A -85,B 0,C 180,E1 18579.661,E2 18579.661} C_VEL
LIN {X 0,Y 246.321,Z 1009.9,A -85,B 0,C 180,E1 18586.859,E2 18586.859} C_VEL
LIN {X 0,Y 234.869,Z 1032.615,A -85,B 0,C 180,E1 18595.499,E2 18595.499} C_VEL
LIN {X 0,Y 227.617,Z 1050.801,A -85,B 0,C 180,E1 18605.558,E2 18605.558} C_VEL
LIN {X 0,Y 225.194,Z 1062.59,A -85,B 0,C 180,E1 18615.556,E2 18615.556} C_VEL
LIN {X 0,Y 225.07,Z 1067.207,A -85,B 0,C 180,E1 18622.268,E2 18622.268} C_VEL
LIN {X 0,Y 225.73,Z 1069.261,A -85,B 0,C 180,E1 18630,E2 18630} C_VEL
LIN {X 0,Y 225.063,Z 1067.215,A -85,B 0,C 180,E1 18637.732,E2 18637.732} C_VEL
LIN {X 0,Y 225.329,Z 1061.489,A -85,B 0,C 180,E1 18645.59,E2 18645.59} C_VEL
LIN {X 0,Y 228.054,Z 1049.589,A -85,B 0,C 180,E1 18655.306,E2 18655.306} C_VEL
LIN {X 0,Y 235.67,Z 1030.891,A -85,B 0,C 180,E1 18665.322,E2 18665.322} C_VEL
LIN {X 0,Y 248.702,Z 1005.772,A -85,B 0,C 180,E1 18674.432,E2 18674.432} C_VEL
LIN {X 0,Y 264.474,Z 976.45,A -85,B 0,C 180,E1 18681.718,E2 18681.718} C_VEL
LIN {X 0,Y 281.393,Z 943.33,A -85,B 0,C 180,E1 18687.341,E2 18687.341} C_VEL
LIN {X 0,Y 297.385,Z 907.867,A -85,B 0,C 180,E1 18691.425,E2 18691.425} C_VEL
LIN {X 0,Y 307.876,Z 879.99,A -85,B 0,C 180,E1 18693.726,E2 18693.726} C_VEL
LIN {X 0,Y 302.824,Z 857.979,A -85,B 0,C 180,E1 18699.126,E2 18699.126} C_VEL
LIN {X 0,Y 296.531,Z 839.458,A -85,B 0,C 180,E1 18705.203,E2 18705.203} C_VEL
LIN {X 0,Y 290.802,Z 825.878,A -85,B 0,C 180,E1 18711.761,E2 18711.761} C_VEL
LIN {X 0,Y 287.828,Z 819.724,A -85,B 0,C 180,E1 18716.545,E2 18716.545} C_VEL
LIN {X 0,Y 286.752,Z 817.222,A -85,B 0,C 180,E1 18719.196,E2 18719.196} C_VEL
LIN {X 0,Y 285.518,Z 817.507,A -85,B 0,C 180,E1 18721.811,E2 18721.811} C_VEL
LIN {X 0,Y 283.24,Z 822.292,A -85,B 0,C 180,E1 18726.199,E2 18726.199} C_VEL
LIN {X 0,Y 284.388,Z 829.835,A -85,B 0,C 180,E1 18735.428,E2 18735.428} C_VEL
LIN {X 0,Y 287.487,Z 840.95,A -85,B 0,C 180,E1 18742.435,E2 18742.435} C_VEL
LIN {X 0,Y 290.675,Z 856.06,A -85,B 0,C 180,E1 18748.849,E2 18748.849} C_VEL
LIN {X 0,Y 292.627,Z 873.595,A -85,B 0,C 180,E1 18754.676,E2 18754.676} C_VEL
LIN {X 0,Y 292.476,Z 884.396,A -85,B 0,C 180,E1 18757.762,E2 18757.762} C_VEL
LIN {X 0,Y 277.486,Z 912.389,A -85,B 0,C 180,E1 18761.979,E2 18761.979} C_VEL
LIN {X 0,Y 261.006,Z 937.865,A -85,B 0,C 180,E1 18767.599,E2 18767.599} C_VEL
LIN {X 0,Y 246.218,Z 957.892,A -85,B 0,C 180,E1 18774.257,E2 18774.257} C_VEL
LIN {X 0,Y 233.916,Z 973.26,A -85,B 0,C 180,E1 18782.082,E2 18782.082} C_VEL
LIN {X 0,Y 225.542,Z 983.549,A -85,B 0,C 180,E1 18790.389,E2 18790.389} C_VEL
LIN {X 0,Y 221.177,Z 989.143,A -85,B 0,C 180,E1 18798.15,E2 18798.15} C_VEL
LIN {X 0,Y 219.389,Z 991.849,A -85,B 0,C 180,E1 18806.043,E2 18806.043} C_VEL
LIN {X 0,Y 219.404,Z 991.818,A -85,B 0,C 180,E1 18813.957,E2 18813.957} C_VEL
LIN {X 0,Y 222.085,Z 987.968,A -85,B 0,C 180,E1 18823.804,E2 18823.804} C_VEL
LIN {X 0,Y 228.864,Z 979.349,A -85,B 0,C 180,E1 18833.386,E2 18833.386} C_VEL
LIN {X 0,Y 240.359,Z 965.146,A -85,B 0,C 180,E1 18842.372,E2 18842.372} C_VEL
LIN {X 0,Y 255.199,Z 945.801,A -85,B 0,C 180,E1 18849.972,E2 18849.972} C_VEL
LIN {X 0,Y 271.008,Z 922.643,A -85,B 0,C 180,E1 18855.923,E2 18855.923} C_VEL
LIN {X 0,Y 286.759,Z 895.45,A -85,B 0,C 180,E1 18860.646,E2 18860.646} C_VEL
LIN {X 0,Y 292.571,Z 883.828,A -85,B 0,C 180,E1 18862.216,E2 18862.216} C_VEL
LIN {X 0,Y 291.785,Z 864.375,A -85,B 0,C 180,E1 18868.104,E2 18868.104} C_VEL
LIN {X 0,Y 288.909,Z 847.49,A -85,B 0,C 180,E1 18874.395,E2 18874.395} C_VEL
LIN {X 0,Y 285.906,Z 835.516,A -85,B 0,C 180,E1 18880.424,E2 18880.424} C_VEL
LIN {X 0,Y 283.774,Z 827.671,A -85,B 0,C 180,E1 18886.122,E2 18886.122} C_VEL
LIN {X 0,Y 283.05,Z 822.039,A -85,B 0,C 180,E1 18893.867,E2 18893.867} C_VEL
LIN {X 0,Y 283.399,Z 822.043,A -85,B 0,C 180,E1 18896.946,E2 18896.946} C_VEL
LIN {X 0,Y 285.83,Z 827.932,A -85,B 0,C 180,E1 18904.565,E2 18904.565} C_VEL
LIN {X 0,Y 290.807,Z 840.675,A -85,B 0,C 180,E1 18912.027,E2 18912.027} C_VEL
LIN {X 0,Y 296.397,Z 856.913,A -85,B 0,C 180,E1 18918.238,E2 18918.238} C_VEL
LIN {X 0,Y 301.577,Z 878.131,A -85,B 0,C 180,E1 18924.116,E2 18924.116} C_VEL
LIN {X 0,Y 302.1,Z 883.995,A -85,B 0,C 180,E1 18925.324,E2 18925.324} C_VEL
LIN {X 0,Y 285.795,Z 923.186,A -85,B 0,C 180,E1 18928.905,E2 18928.905} C_VEL
LIN {X 0,Y 268.329,Z 958.261,A -85,B 0,C 180,E1 18933.753,E2 18933.753} C_VEL
LIN {X 0,Y 251.587,Z 988.511,A -85,B 0,C 180,E1 18939.891,E2 18939.891} C_VEL
LIN {X 0,Y 235.801,Z 1016.332,A -85,B 0,C 180,E1 18948.206,E2 18948.206} C_VEL
LIN {X 0,Y 224.929,Z 1037.425,A -85,B 0,C 180,E1 18957.42,E2 18957.42} C_VEL
LIN {X 0,Y 218.83,Z 1053.371,A -85,B 0,C 180,E1 18967.634,E2 18967.634} C_VEL
LIN {X 0,Y 217.269,Z 1062.963,A -85,B 0,C 180,E1 18977.333,E2 18977.333} C_VEL
LIN {X 0,Y 217.461,Z 1067.333,A -85,B 0,C 180,E1 18986.007,E2 18986.007} C_VEL
LIN {X 0,Y 217.956,Z 1067.915,A -85,B 0,C 180,E1 18990,E2 18990} C_VEL
LIN {X 0,Y 217.227,Z 1065.843,A -85,B 0,C 180,E1 18998.012,E2 18998.012} C_VEL
LIN {X 0,Y 217.532,Z 1060.08,A -85,B 0,C 180,E1 19006.164,E2 19006.164} C_VEL
LIN {X 0,Y 220.326,Z 1048.821,A -85,B 0,C 180,E1 19015.746,E2 19015.746} C_VEL
LIN {X 0,Y 228.85,Z 1029.399,A -85,B 0,C 180,E1 19026.541,E2 19026.541} C_VEL
LIN {X 0,Y 242.437,Z 1004.792,A -85,B 0,C 180,E1 19035.664,E2 19035.664} C_VEL
LIN {X 0,Y 259.431,Z 974.525,A -85,B 0,C 180,E1 19043.264,E2 19043.264} C_VEL
LIN {X 0,Y 276.951,Z 941.644,A -85,B 0,C 180,E1 19048.804,E2 19048.804} C_VEL
LIN {X 0,Y 293.471,Z 906.116,A -85,B 0,C 180,E1 19052.839,E2 19052.839} C_VEL
LIN {X 0,Y 302.454,Z 882.906,A -85,B 0,C 180,E1 19054.811,E2 19054.811} C_VEL
LIN {X 0,Y 297.838,Z 861.683,A -85,B 0,C 180,E1 19060.314,E2 19060.314} C_VEL
LIN {X 0,Y 292.206,Z 844.001,A -85,B 0,C 180,E1 19066.51,E2 19066.51} C_VEL
LIN {X 0,Y 287.349,Z 832.137,A -85,B 0,C 180,E1 19072.804,E2 19072.804} C_VEL
LIN {X 0,Y 285.116,Z 826.93,A -85,B 0,C 180,E1 19076.948,E2 19076.948} C_VEL
LIN {X 0,Y 283.651,Z 822.072,A -85,B 0,C 180,E1 19083.051,E2 19083.051} C_VEL
LIN {X 0,Y 283.24,Z 822.292,A -85,B 0,C 180,E1 19086.199,E2 19086.199} C_VEL
LIN {X 0,Y 281.771,Z 828.24,A -85,B 0,C 180,E1 19089.524,E2 19089.524} C_VEL
LIN {X 0,Y 280.743,Z 834.618,A -85,B 0,C 180,E1 19092.861,E2 19092.861} C_VEL
LIN {X 0,Y 282.757,Z 843.159,A -85,B 0,C 180,E1 19099.541,E2 19099.541} C_VEL
LIN {X 0,Y 285.293,Z 855.736,A -85,B 0,C 180,E1 19105.819,E2 19105.819} C_VEL
LIN {X 0,Y 287.188,Z 872.779,A -85,B 0,C 180,E1 19112.175,E2 19112.175} C_VEL
LIN {X 0,Y 286.936,Z 887.7,A -85,B 0,C 180,E1 19116.766,E2 19116.766} C_VEL
LIN {X 0,Y 271.212,Z 915.669,A -85,B 0,C 180,E1 19121.096,E2 19121.096} C_VEL
LIN {X 0,Y 254.327,Z 940.628,A -85,B 0,C 180,E1 19126.797,E2 19126.797} C_VEL
LIN {X 0,Y 238.328,Z 961.249,A -85,B 0,C 180,E1 19134.013,E2 19134.013} C_VEL
LIN {X 0,Y 224.789,Z 977.277,A -85,B 0,C 180,E1 19142.96,E2 19142.96} C_VEL
LIN {X 0,Y 215.538,Z 988.07,A -85,B 0,C 180,E1 19153.682,E2 19153.682} C_VEL
LIN {X 0,Y 212.22,Z 992.2,A -85,B 0,C 180,E1 19161.797,E2 19161.797} C_VEL
LIN {X 0,Y 211.666,Z 993.499,A -85,B 0,C 180,E1 19170,E2 19170} C_VEL
LIN {X 0,Y 212.249,Z 992.149,A -85,B 0,C 180,E1 19178.202,E2 19178.202} C_VEL
LIN {X 0,Y 216.79,Z 986.462,A -85,B 0,C 180,E1 19188.317,E2 19188.317} C_VEL
LIN {X 0,Y 226.019,Z 975.723,A -85,B 0,C 180,E1 19197.963,E2 19197.963} C_VEL
LIN {X 0,Y 238.459,Z 960.998,A -85,B 0,C 180,E1 19205.965,E2 19205.965} C_VEL
LIN {X 0,Y 254.45,Z 940.293,A -85,B 0,C 180,E1 19213.177,E2 19213.177} C_VEL
LIN {X 0,Y 271.299,Z 915.245,A -85,B 0,C 180,E1 19218.884,E2 19218.884} C_VEL
LIN {X 0,Y 286.996,Z 887.324,A -85,B 0,C 180,E1 19223.165,E2 19223.165} C_VEL
LIN {X 0,Y 286.756,Z 868.471,A -85,B 0,C 180,E1 19229.142,E2 19229.142} C_VEL
LIN {X 0,Y 284.508,Z 852.263,A -85,B 0,C 180,E1 19235.567,E2 19235.567} C_VEL
LIN {X 0,Y 281.958,Z 840.251,A -85,B 0,C 180,E1 19242.127,E2 19242.127} C_VEL
LIN {X 0,Y 280.472,Z 833.957,A -85,B 0,C 180,E1 19247.54,E2 19247.54} C_VEL
LIN {X 0,Y 280.487,Z 829.591,A -85,B 0,C 180,E1 19253.811,E2 19253.811} C_VEL
LIN {X 0,Y 280.859,Z 829.55,A -85,B 0,C 180,E1 19256.918,E2 19256.918} C_VEL
LIN {X 0,Y 283.151,Z 835.703,A -85,B 0,C 180,E1 19264.608,E2 19264.608} C_VEL
LIN {X 0,Y 287.782,Z 848.581,A -85,B 0,C 180,E1 19272.155,E2 19272.155} C_VEL
LIN {X 0,Y 292.803,Z 865.211,A -85,B 0,C 180,E1 19278.424,E2 19278.424} C_VEL
LIN {X 0,Y 296.966,Z 885.702,A -85,B 0,C 180,E1 19284.076,E2 19284.076} C_VEL
LIN {X 0,Y 280.341,Z 924.538,A -85,B 0,C 180,E1 19287.778,E2 19287.778} C_VEL
LIN {X 0,Y 262.415,Z 958.968,A -85,B 0,C 180,E1 19292.632,E2 19292.632} C_VEL
LIN {X 0,Y 245.143,Z 988.735,A -85,B 0,C 180,E1 19298.832,E2 19298.832} C_VEL
LIN {X 0,Y 229.563,Z 1014.837,A -85,B 0,C 180,E1 19306.805,E2 19306.805} C_VEL
LIN {X 0,Y 217.558,Z 1036.665,A -85,B 0,C 180,E1 19316.636,E2 19316.636} C_VEL
LIN {X 0,Y 211.247,Z 1051.937,A -85,B 0,C 180,E1 19326.785,E2 19326.785} C_VEL
LIN {X 0,Y 209.537,Z 1060.465,A -85,B 0,C 180,E1 19335.351,E2 19335.351} C_VEL
LIN {X 0,Y 209.395,Z 1064.461,A -85,B 0,C 180,E1 19341.685,E2 19341.685} C_VEL
LIN {X 0,Y 210.151,Z 1066.563,A -85,B 0,C 180,E1 19350,E2 19350} C_VEL
LIN {X 0,Y 209.389,Z 1064.47,A -85,B 0,C 180,E1 19358.314,E2 19358.314} C_VEL
LIN {X 0,Y 209.737,Z 1058.668,A -85,B 0,C 180,E1 19366.782,E2 19366.782} C_VEL
LIN {X 0,Y 213.273,Z 1046.404,A -85,B 0,C 180,E1 19377.398,E2 19377.398} C_VEL
LIN {X 0,Y 222.147,Z 1027.905,A -85,B 0,C 180,E1 19387.833,E2 19387.833} C_VEL
LIN {X 0,Y 237.111,Z 1002.281,A -85,B 0,C 180,E1 19397.431,E2 19397.431} C_VEL
LIN {X 0,Y 254.638,Z 972.674,A -85,B 0,C 180,E1 19404.838,E2 19404.838} C_VEL
LIN {X 0,Y 272.372,Z 940.597,A -85,B 0,C 180,E1 19410.226,E2 19410.226} C_VEL
LIN {X 0,Y 289.357,Z 905.273,A -85,B 0,C 180,E1 19414.209,E2 19414.209} C_VEL
LIN {X 0,Y 297.05,Z 885.804,A -85,B 0,C 180,E1 19415.931,E2 19415.931} C_VEL
LIN {X 0,Y 292.951,Z 865.414,A -85,B 0,C 180,E1 19421.552,E2 19421.552} C_VEL
LIN {X 0,Y 287.934,Z 848.693,A -85,B 0,C 180,E1 19427.852,E2 19427.852} C_VEL
LIN {X 0,Y 283.294,Z 835.927,A -85,B 0,C 180,E1 19435.394,E2 19435.394} C_VEL
LIN {X 0,Y 281.115,Z 829.571,A -85,B 0,C 180,E1 19443.079,E2 19443.079} C_VEL
LIN {X 0,Y 280.445,Z 830.587,A -85,B 0,C 180,E1 19447.426,E2 19447.426} C_VEL
LIN {X 0,Y 280.743,Z 834.618,A -85,B 0,C 180,E1 19452.861,E2 19452.861} C_VEL
LIN {X 0,Y 280.391,Z 839.527,A -85,B 0,C 180,E1 19455.343,E2 19455.343} C_VEL
LIN {X 0,Y 279.175,Z 850.184,A -85,B 0,C 180,E1 19459.334,E2 19459.334} C_VEL
LIN {X 0,Y 281,Z 862.281,A -85,B 0,C 180,E1 19465.522,E2 19465.522} C_VEL
LIN {X 0,Y 282.116,Z 879.272,A -85,B 0,C 180,E1 19472.019,E2 19472.019} C_VEL
LIN {X 0,Y 281.156,Z 891.619,A -85,B 0,C 180,E1 19475.806,E2 19475.806} C_VEL
LIN {X 0,Y 263.899,Z 920.744,A -85,B 0,C 180,E1 19480.523,E2 19480.523} C_VEL
LIN {X 0,Y 245.696,Z 945.977,A -85,B 0,C 180,E1 19486.723,E2 19486.723} C_VEL
LIN {X 0,Y 230.423,Z 964.555,A -85,B 0,C 180,E1 19493.748,E2 19493.748} C_VEL
LIN {X 0,Y 216.703,Z 979.847,A -85,B 0,C 180,E1 19502.992,E2 19502.992} C_VEL
LIN {X 0,Y 208.052,Z 989.422,A -85,B 0,C 180,E1 19513.078,E2 19513.078} C_VEL
LIN {X 0,Y 204.513,Z 993.55,A -85,B 0,C 180,E1 19521.486,E2 19521.486} C_VEL
LIN {X 0,Y 203.903,Z 994.844,A -85,B 0,C 180,E1 19530,E2 19530} C_VEL
LIN {X 0,Y 204.542,Z 993.497,A -85,B 0,C 180,E1 19538.513,E2 19538.513} C_VEL
LIN {X 0,Y 209.377,Z 987.821,A -85,B 0,C 180,E1 19548.99,E2 19548.99} C_VEL
LIN {X 0,Y 219.163,Z 977.086,A -85,B 0,C 180,E1 19558.919,E2 19558.919} C_VEL
LIN {X 0,Y 232.185,Z 962.377,A -85,B 0,C 180,E1 19567.097,E2 19567.097} C_VEL
LIN {X 0,Y 248.83,Z 941.704,A -85,B 0,C 180,E1 19574.404,E2 19574.404} C_VEL
LIN {X 0,Y 266.268,Z 916.718,A -85,B 0,C 180,E1 19580.14,E2 19580.14} C_VEL
LIN {X 0,Y 281.558,Z 889.951,A -85,B 0,C 180,E1 19584.419,E2 19584.419} C_VEL
LIN {X 0,Y 281.818,Z 872.761,A -85,B 0,C 180,E1 19590.153,E2 19590.153} C_VEL
LIN {X 0,Y 280.216,Z 857.176,A -85,B 0,C 180,E1 19596.708,E2 19596.708} C_VEL
LIN {X 0,Y 278.264,Z 845.859,A -85,B 0,C 180,E1 19603.413,E2 19603.413} C_VEL
LIN {X 0,Y 277.34,Z 838.397,A -85,B 0,C 180,E1 19611.33,E2 19611.33} C_VEL
LIN {X 0,Y 278.047,Z 836.944,A -85,B 0,C 180,E1 19616.887,E2 19616.887} C_VEL
LIN {X 0,Y 280.181,Z 843.338,A -85,B 0,C 180,E1 19624.657,E2 19624.657} C_VEL
LIN {X 0,Y 284.012,Z 854.866,A -85,B 0,C 180,E1 19631.538,E2 19631.538} C_VEL
LIN {X 0,Y 288.209,Z 870.33,A -85,B 0,C 180,E1 19637.588,E2 19637.588} C_VEL
LIN {X 0,Y 291.559,Z 888.634,A -85,B 0,C 180,E1 19642.927,E2 19642.927} C_VEL
LIN {X 0,Y 275.571,Z 924.75,A -85,B 0,C 180,E1 19646.472,E2 19646.472} C_VEL
LIN {X 0,Y 257.122,Z 958.848,A -85,B 0,C 180,E1 19651.324,E2 19651.324} C_VEL
LIN {X 0,Y 239.643,Z 987.648,A -85,B 0,C 180,E1 19657.38,E2 19657.38} C_VEL
LIN {X 0,Y 222.648,Z 1014.579,A -85,B 0,C 180,E1 19665.801,E2 19665.801} C_VEL
LIN {X 0,Y 210.36,Z 1035.591,A -85,B 0,C 180,E1 19675.612,E2 19675.612} C_VEL
LIN {X 0,Y 203.713,Z 1050.503,A -85,B 0,C 180,E1 19685.873,E2 19685.873} C_VEL
LIN {X 0,Y 201.596,Z 1060.63,A -85,B 0,C 180,E1 19696.979,E2 19696.979} C_VEL
LIN {X 0,Y 201.806,Z 1064.612,A -85,B 0,C 180,E1 19705.697,E2 19705.697} C_VEL
LIN {X 0,Y 202.374,Z 1065.216,A -85,B 0,C 180,E1 19710,E2 19710} C_VEL
LIN {X 0,Y 201.553,Z 1063.097,A -85,B 0,C 180,E1 19718.64,E2 19718.64} C_VEL
LIN {X 0,Y 201.961,Z 1057.254,A -85,B 0,C 180,E1 19727.449,E2 19727.449} C_VEL
LIN {X 0,Y 205.553,Z 1045.779,A -85,B 0,C 180,E1 19737.874,E2 19737.874} C_VEL
LIN {X 0,Y 215.525,Z 1026.406,A -85,B 0,C 180,E1 19749.214,E2 19749.214} C_VEL
LIN {X 0,Y 230.847,Z 1001.651,A -85,B 0,C 180,E1 19758.712,E2 19758.712} C_VEL
LIN {X 0,Y 248.736,Z 973.01,A -85,B 0,C 180,E1 19766.028,E2 19766.028} C_VEL
LIN {X 0,Y 268.053,Z 939.416,A -85,B 0,C 180,E1 19771.713,E2 19771.713} C_VEL
LIN {X 0,Y 285.849,Z 903.44,A -85,B 0,C 180,E1 19775.704,E2 19775.704} C_VEL
LIN {X 0,Y 291.66,Z 888.832,A -85,B 0,C 180,E1 19777.057,E2 19777.057} C_VEL
LIN {X 0,Y 288.09,Z 869.287,A -85,B 0,C 180,E1 19782.799,E2 19782.799} C_VEL
LIN {X 0,Y 284.157,Z 854.985,A -85,B 0,C 180,E1 19788.468,E2 19788.468} C_VEL
LIN {X 0,Y 280.302,Z 843.611,A -85,B 0,C 180,E1 19795.345,E2 19795.345} C_VEL
LIN {X 0,Y 278.3,Z 836.966,A -85,B 0,C 180,E1 19803.11,E2 19803.11} C_VEL
LIN {X 0,Y 277.552,Z 838.083,A -85,B 0,C 180,E1 19807.504,E2 19807.504} C_VEL
LIN {X 0,Y 278.213,Z 845.173,A -85,B 0,C 180,E1 19815.779,E2 19815.779} C_VEL
LIN {X 0,Y 279.175,Z 850.184,A -85,B 0,C 180,E1 19819.334,E2 19819.334} C_VEL
LIN {X 0,Y 278.738,Z 856.535,A -85,B 0,C 180,E1 19821.688,E2 19821.688} C_VEL
LIN {X 0,Y 276.658,Z 869.264,A -85,B 0,C 180,E1 19825.431,E2 19825.431} C_VEL
LIN {X 0,Y 276.923,Z 885.837,A -85,B 0,C 180,E1 19831.875,E2 19831.875} C_VEL
LIN {X 0,Y 276.06,Z 894.358,A -85,B 0,C 180,E1 19834.65,E2 19834.65} C_VEL
LIN {X 0,Y 257.73,Z 923.86,A -85,B 0,C 180,E1 19839.556,E2 19839.556} C_VEL
LIN {X 0,Y 239.051,Z 948.6,A -85,B 0,C 180,E1 19845.84,E2 19845.84} C_VEL
LIN {X 0,Y 222.511,Z 967.697,A -85,B 0,C 180,E1 19853.462,E2 19853.462} C_VEL
LIN {X 0,Y 208.605,Z 982.393,A -85,B 0,C 180,E1 19863.025,E2 19863.025} C_VEL
LIN {X 0,Y 199.381,Z 992.121,A -85,B 0,C 180,E1 19874.588,E2 19874.588} C_VEL
LIN {X 0,Y 196.095,Z 995.894,A -85,B 0,C 180,E1 19885.572,E2 19885.572} C_VEL
LIN {X 0,Y 196.133,Z 995.86,A -85,B 0,C 180,E1 19894.427,E2 19894.427} C_VEL
LIN {X 0,Y 199.405,Z 992.035,A -85,B 0,C 180,E1 19905.411,E2 19905.411} C_VEL
LIN {X 0,Y 207.563,Z 983.432,A -85,B 0,C 180,E1 19915.954,E2 19915.954} C_VEL
LIN {X 0,Y 220.967,Z 969.26,A -85,B 0,C 180,E1 19925.619,E2 19925.619} C_VEL
LIN {X 0,Y 237.857,Z 949.899,A -85,B 0,C 180,E1 19933.619,E2 19933.619} C_VEL
LIN {X 0,Y 255.882,Z 926.227,A -85,B 0,C 180,E1 19939.841,E2 19939.841} C_VEL
LIN {X 0,Y 273.305,Z 898.914,A -85,B 0,C 180,E1 19944.578,E2 19944.578} C_VEL
LIN {X 0,Y 276.233,Z 892.808,A -85,B 0,C 180,E1 19945.652,E2 19945.652} C_VEL
LIN {X 0,Y 276.874,Z 875.81,A -85,B 0,C 180,E1 19951.696,E2 19951.696} C_VEL
LIN {X 0,Y 275.792,Z 861.322,A -85,B 0,C 180,E1 19958.261,E2 19958.261} C_VEL
LIN {X 0,Y 274.464,Z 850.497,A -85,B 0,C 180,E1 19965.637,E2 19965.637} C_VEL
LIN {X 0,Y 274.608,Z 844.416,A -85,B 0,C 180,E1 19973.678,E2 19973.678} C_VEL
LIN {X 0,Y 275.131,Z 844.305,A -85,B 0,C 180,E1 19976.854,E2 19976.854} C_VEL
LIN {X 0,Y 277.057,Z 850.91,A -85,B 0,C 180,E1 19984.71,E2 19984.71} C_VEL
LIN {X 0,Y 280.633,Z 862.641,A -85,B 0,C 180,E1 19991.679,E2 19991.679} C_VEL
LIN {X 0,Y 284.274,Z 878.62,A -85,B 0,C 180,E1 19997.839,E2 19997.839} C_VEL
LIN {X 0,Y 286,Z 893.511,A -85,B 0,C 180,E1 20002.075,E2 20002.075} C_VEL
LIN {X 0,Y 267.446,Z 931.666,A -85,B 0,C 180,E1 20005.915,E2 20005.915} C_VEL
LIN {X 0,Y 247.774,Z 965.544,A -85,B 0,C 180,E1 20011.19,E2 20011.19} C_VEL
LIN {X 0,Y 228.724,Z 994.866,A -85,B 0,C 180,E1 20018.098,E2 20018.098} C_VEL
LIN {X 0,Y 211.913,Z 1020.341,A -85,B 0,C 180,E1 20027.256,E2 20027.256} C_VEL
LIN {X 0,Y 200.216,Z 1040.097,A -85,B 0,C 180,E1 20038.04,E2 20038.04} C_VEL
LIN {X 0,Y 194.804,Z 1053.218,A -85,B 0,C 180,E1 20048.868,E2 20048.868} C_VEL
LIN {X 0,Y 193.749,Z 1060.857,A -85,B 0,C 180,E1 20059.276,E2 20059.276} C_VEL
LIN {X 0,Y 193.98,Z 1063.252,A -85,B 0,C 180,E1 20065.523,E2 20065.523} C_VEL
LIN {X 0,Y 194.564,Z 1063.863,A -85,B 0,C 180,E1 20070,E2 20070} C_VEL
LIN {X 0,Y 193.723,Z 1061.723,A -85,B 0,C 180,E1 20078.992,E2 20078.992} C_VEL
LIN {X 0,Y 194.476,Z 1054.559,A -85,B 0,C 180,E1 20089.655,E2 20089.655} C_VEL
LIN {X 0,Y 199.732,Z 1041.206,A -85,B 0,C 180,E1 20101.214,E2 20101.214} C_VEL
LIN {X 0,Y 211.187,Z 1021.53,A -85,B 0,C 180,E1 20112.228,E2 20112.228} C_VEL
LIN {X 0,Y 226.999,Z 997.576,A -85,B 0,C 180,E1 20121.11,E2 20121.11} C_VEL
LIN {X 0,Y 245.311,Z 969.507,A -85,B 0,C 180,E1 20128.061,E2 20128.061} C_VEL
LIN {X 0,Y 264.44,Z 937.281,A -85,B 0,C 180,E1 20133.374,E2 20133.374} C_VEL
LIN {X 0,Y 282.482,Z 901.698,A -85,B 0,C 180,E1 20137.236,E2 20137.236} C_VEL
LIN {X 0,Y 286.405,Z 892.509,A -85,B 0,C 180,E1 20138.072,E2 20138.072} C_VEL
LIN {X 0,Y 283.409,Z 873.976,A -85,B 0,C 180,E1 20143.786,E2 20143.786} C_VEL
LIN {X 0,Y 279.837,Z 859.69,A -85,B 0,C 180,E1 20149.865,E2 20149.865} C_VEL
LIN {X 0,Y 276.584,Z 849.379,A -85,B 0,C 180,E1 20156.854,E2 20156.854} C_VEL
LIN {X 0,Y 275.381,Z 844.33,A -85,B 0,C 180,E1 20163.143,E2 20163.143} C_VEL
LIN {X 0,Y 274.575,Z 845.135,A -85,B 0,C 180,E1 20167.019,E2 20167.019} C_VEL
LIN {X 0,Y 274.638,Z 850.743,A -85,B 0,C 180,E1 20174.354,E2 20174.354} C_VEL
LIN {X 0,Y 275.824,Z 860.437,A -85,B 0,C 180,E1 20181.073,E2 20181.073} C_VEL
LIN {X 0,Y 276.658,Z 869.264,A -85,B 0,C 180,E1 20185.431,E2 20185.431} C_VEL
LIN {X 0,Y 275.507,Z 876.716,A -85,B 0,C 180,E1 20187.658,E2 20187.658} C_VEL
LIN {X 0,Y 271.629,Z 890.694,A -85,B 0,C 180,E1 20191.195,E2 20191.195} C_VEL
LIN {X 0,Y 270.806,Z 897.447,A -85,B 0,C 180,E1 20193.525,E2 20193.525} C_VEL
LIN {X 0,Y 252.85,Z 925.298,A -85,B 0,C 180,E1 20198.198,E2 20198.198} C_VEL
LIN {X 0,Y 233.527,Z 949.992,A -85,B 0,C 180,E1 20204.509,E2 20204.509} C_VEL
LIN {X 0,Y 216.283,Z 969.064,A -85,B 0,C 180,E1 20212.23,E2 20212.23} C_VEL
LIN {X 0,Y 201.674,Z 983.752,A -85,B 0,C 180,E1 20222.018,E2 20222.018} C_VEL
LIN {X 0,Y 191.854,Z 993.476,A -85,B 0,C 180,E1 20233.967,E2 20233.967} C_VEL
LIN {X 0,Y 188.345,Z 997.241,A -85,B 0,C 180,E1 20245.39,E2 20245.39} C_VEL
LIN {X 0,Y 188.382,Z 997.207,A -85,B 0,C 180,E1 20254.61,E2 20254.61} C_VEL
LIN {X 0,Y 191.881,Z 993.391,A -85,B 0,C 180,E1 20266.031,E2 20266.031} C_VEL
LIN {X 0,Y 200.563,Z 984.794,A -85,B 0,C 180,E1 20276.932,E2 20276.932} C_VEL
LIN {X 0,Y 214.669,Z 970.635,A -85,B 0,C 180,E1 20286.833,E2 20286.833} C_VEL
LIN {X 0,Y 232.651,Z 950.873,A -85,B 0,C 180,E1 20295.077,E2 20295.077} C_VEL
LIN {X 0,Y 251.735,Z 926.575,A -85,B 0,C 180,E1 20301.431,E2 20301.431} C_VEL
LIN {X 0,Y 270.225,Z 898.198,A -85,B 0,C 180,E1 20306.243,E2 20306.243} C_VEL
LIN {X 0,Y 271.881,Z 884.587,A -85,B 0,C 180,E1 20310.977,E2 20310.977} C_VEL
LIN {X 0,Y 271.756,Z 870.853,A -85,B 0,C 180,E1 20317.058,E2 20317.058} C_VEL
LIN {X 0,Y 271.068,Z 859.901,A -85,B 0,C 180,E1 20323.794,E2 20323.794} C_VEL
LIN {X 0,Y 270.938,Z 853.072,A -85,B 0,C 180,E1 20331.357,E2 20331.357} C_VEL
LIN {X 0,Y 271.935,Z 851.541,A -85,B 0,C 180,E1 20336.817,E2 20336.817} C_VEL
LIN {X 0,Y 273.763,Z 858.369,A -85,B 0,C 180,E1 20344.766,E2 20344.766} C_VEL
LIN {X 0,Y 276.902,Z 870.438,A -85,B 0,C 180,E1 20351.839,E2 20351.839} C_VEL
LIN {X 0,Y 279.942,Z 886.957,A -85,B 0,C 180,E1 20358.125,E2 20358.125} C_VEL
LIN {X 0,Y 280.995,Z 895.725,A -85,B 0,C 180,E1 20360.795,E2 20360.795} C_VEL
LIN {X 0,Y 262.329,Z 932.731,A -85,B 0,C 180,E1 20364.634,E2 20364.634} C_VEL
LIN {X 0,Y 242.866,Z 964.992,A -85,B 0,C 180,E1 20369.704,E2 20369.704} C_VEL
LIN {X 0,Y 222.974,Z 994.235,A -85,B 0,C 180,E1 20376.665,E2 20376.665} C_VEL
LIN {X 0,Y 205.759,Z 1018.839,A -85,B 0,C 180,E1 20385.652,E2 20385.652} C_VEL
LIN {X 0,Y 193.177,Z 1038.639,A -85,B 0,C 180,E1 20396.728,E2 20396.728} C_VEL
LIN {X 0,Y 187.142,Z 1051.782,A -85,B 0,C 180,E1 20407.958,E2 20407.958} C_VEL
LIN {X 0,Y 185.889,Z 1058.98,A -85,B 0,C 180,E1 20417.818,E2 20417.818} C_VEL
LIN {X 0,Y 186.152,Z 1061.891,A -85,B 0,C 180,E1 20425.335,E2 20425.335} C_VEL
LIN {X 0,Y 186.783,Z 1062.515,A -85,B 0,C 180,E1 20430,E2 20430} C_VEL
LIN {X 0,Y 185.9,Z 1060.349,A -85,B 0,C 180,E1 20439.374,E2 20439.374} C_VEL
LIN {X 0,Y 186.79,Z 1053.138,A -85,B 0,C 180,E1 20450.499,E2 20450.499} C_VEL
LIN {X 0,Y 192.324,Z 1040.311,A -85,B 0,C 180,E1 20462.096,E2 20462.096} C_VEL
LIN {X 0,Y 204.203,Z 1021.161,A -85,B 0,C 180,E1 20473.299,E2 20473.299} C_VEL
LIN {X 0,Y 221.432,Z 996.522,A -85,B 0,C 180,E1 20482.671,E2 20482.671} C_VEL
LIN {X 0,Y 241.418,Z 967.282,A -85,B 0,C 180,E1 20489.879,E2 20489.879} C_VEL
LIN {X 0,Y 261.636,Z 934.175,A -85,B 0,C 180,E1 20495.199,E2 20495.199} C_VEL
LIN {X 0,Y 280.271,Z 897.975,A -85,B 0,C 180,E1 20498.963,E2 20498.963} C_VEL
LIN {X 0,Y 281.027,Z 895.237,A -85,B 0,C 180,E1 20499.392,E2 20499.392} C_VEL
LIN {X 0,Y 278.563,Z 877.577,A -85,B 0,C 180,E1 20505.233,E2 20505.233} C_VEL
LIN {X 0,Y 275.52,Z 864.559,A -85,B 0,C 180,E1 20511.28,E2 20511.28} C_VEL
LIN {X 0,Y 273.317,Z 856.764,A -85,B 0,C 180,E1 20516.817,E2 20516.817} C_VEL
LIN {X 0,Y 272.174,Z 851.588,A -85,B 0,C 180,E1 20523.18,E2 20523.18} C_VEL
LIN {X 0,Y 271.15,Z 853.105,A -85,B 0,C 180,E1 20528.015,E2 20528.015} C_VEL
LIN {X 0,Y 271.074,Z 858.487,A -85,B 0,C 180,E1 20534.808,E2 20534.808} C_VEL
LIN {X 0,Y 271.803,Z 868.204,A -85,B 0,C 180,E1 20541.4,E2 20541.4} C_VEL
LIN {X 0,Y 272.054,Z 882.369,A -85,B 0,C 180,E1 20547.998,E2 20547.998} C_VEL
LIN {X 0,Y 271.629,Z 890.694,A -85,B 0,C 180,E1 20551.195,E2 20551.195} C_VEL
LIN {X 0,Y 268.953,Z 896.772,A -85,B 0,C 180,E1 20552.336,E2 20552.336} C_VEL
LIN {X 0,Y 260.629,Z 908.618,A -85,B 0,C 180,E1 20553.549,E2 20553.549} C_VEL
LIN {X 0,Y 241.77,Z 935.089,A -85,B 0,C 180,E1 20558.631,E2 20558.631} C_VEL
LIN {X 0,Y 222.416,Z 957.716,A -85,B 0,C 180,E1 20565.312,E2 20565.312} C_VEL
LIN {X 0,Y 204.929,Z 975.505,A -85,B 0,C 180,E1 20573.77,E2 20573.77} C_VEL
LIN {X 0,Y 191.282,Z 988.362,A -85,B 0,C 180,E1 20584.195,E2 20584.195} C_VEL
LIN {X 0,Y 183.182,Z 995.896,A -85,B 0,C 180,E1 20595.644,E2 20595.644} C_VEL
LIN {X 0,Y 180.576,Z 998.591,A -85,B 0,C 180,E1 20605.191,E2 20605.191} C_VEL
LIN {X 0,Y 180.612,Z 998.558,A -85,B 0,C 180,E1 20614.809,E2 20614.809} C_VEL
LIN {X 0,Y 184.396,Z 994.745,A -85,B 0,C 180,E1 20626.701,E2 20626.701} C_VEL
LIN {X 0,Y 193.63,Z 986.156,A -85,B 0,C 180,E1 20637.979,E2 20637.979} C_VEL
LIN {X 0,Y 208.489,Z 972.002,A -85,B 0,C 180,E1 20648.116,E2 20648.116} C_VEL
LIN {X 0,Y 227.181,Z 952.319,A -85,B 0,C 180,E1 20656.447,E2 20656.447} C_VEL
LIN {X 0,Y 246.964,Z 928.023,A -85,B 0,C 180,E1 20662.84,E2 20662.84} C_VEL
LIN {X 0,Y 265.194,Z 901.06,A -85,B 0,C 180,E1 20667.442,E2 20667.442} C_VEL
LIN {X 0,Y 267.049,Z 886.447,A -85,B 0,C 180,E1 20673.04,E2 20673.04} C_VEL
LIN {X 0,Y 267.303,Z 873.739,A -85,B 0,C 180,E1 20679.279,E2 20679.279} C_VEL
LIN {X 0,Y 267.12,Z 865.319,A -85,B 0,C 180,E1 20685.232,E2 20685.232} C_VEL
LIN {X 0,Y 267.943,Z 858.96,A -85,B 0,C 180,E1 20693.52,E2 20693.52} C_VEL
LIN {X 0,Y 268.596,Z 858.723,A -85,B 0,C 180,E1 20696.777,E2 20696.777} C_VEL
LIN {X 0,Y 270.21,Z 865.717,A -85,B 0,C 180,E1 20704.829,E2 20704.829} C_VEL
LIN {X 0,Y 272.728,Z 876.457,A -85,B 0,C 180,E1 20711.211,E2 20711.211} C_VEL
LIN {X 0,Y 275.165,Z 892.804,A -85,B 0,C 180,E1 20717.622,E2 20717.622} C_VEL
LIN {X 0,Y 275.47,Z 899.81,A -85,B 0,C 180,E1 20719.747,E2 20719.747} C_VEL
LIN {X 0,Y 256.062,Z 935.998,A -85,B 0,C 180,E1 20723.587,E2 20723.587} C_VEL
LIN {X 0,Y 235.924,Z 967.581,A -85,B 0,C 180,E1 20728.759,E2 20728.759} C_VEL
LIN {X 0,Y 215.025,Z 996.691,A -85,B 0,C 180,E1 20736.086,E2 20736.086} C_VEL
LIN {X 0,Y 197.271,Z 1020.848,A -85,B 0,C 180,E1 20745.626,E2 20745.626} C_VEL
LIN {X 0,Y 184.325,Z 1040.405,A -85,B 0,C 180,E1 20757.731,E2 20757.731} C_VEL
LIN {X 0,Y 178.797,Z 1052.986,A -85,B 0,C 180,E1 20770.202,E2 20770.202} C_VEL
LIN {X 0,Y 178.087,Z 1058.962,A -85,B 0,C 180,E1 20780.21,E2 20780.21} C_VEL
LIN {X 0,Y 178.99,Z 1061.166,A -85,B 0,C 180,E1 20790,E2 20790} C_VEL
LIN {X 0,Y 178.079,Z 1058.974,A -85,B 0,C 180,E1 20799.79,E2 20799.79} C_VEL
LIN {X 0,Y 179.193,Z 1051.54,A -85,B 0,C 180,E1 20811.639,E2 20811.639} C_VEL
LIN {X 0,Y 185.266,Z 1038.842,A -85,B 0,C 180,E1 20823.477,E2 20823.477} C_VEL
LIN {X 0,Y 197.944,Z 1019.891,A -85,B 0,C 180,E1 20834.873,E2 20834.873} C_VEL
LIN {X 0,Y 215.866,Z 995.722,A -85,B 0,C 180,E1 20844.232,E2 20844.232} C_VEL
LIN {X 0,Y 236.041,Z 967.572,A -85,B 0,C 180,E1 20851.268,E2 20851.268} C_VEL
LIN {X 0,Y 256.804,Z 934.985,A -85,B 0,C 180,E1 20856.561,E2 20856.561} C_VEL
LIN {X 0,Y 275.779,Z 899.016,A -85,B 0,C 180,E1 20860.426,E2 20860.426} C_VEL
LIN {X 0,Y 273.79,Z 881.962,A -85,B 0,C 180,E1 20866.4,E2 20866.4} C_VEL
LIN {X 0,Y 271.505,Z 870.729,A -85,B 0,C 180,E1 20871.936,E2 20871.936} C_VEL
LIN {X 0,Y 269.33,Z 862.364,A -85,B 0,C 180,E1 20878.542,E2 20878.542} C_VEL
LIN {X 0,Y 268.826,Z 858.78,A -85,B 0,C 180,E1 20883.22,E2 20883.22} C_VEL
LIN {X 0,Y 267.602,Z 860.326,A -85,B 0,C 180,E1 20888.122,E2 20888.122} C_VEL
LIN {X 0,Y 267.283,Z 866.607,A -85,B 0,C 180,E1 20895.647,E2 20895.647} C_VEL
LIN {X 0,Y 267.451,Z 877.221,A -85,B 0,C 180,E1 20902.453,E2 20902.453} C_VEL
LIN {X 0,Y 266.82,Z 891.262,A -85,B 0,C 180,E1 20908.824,E2 20908.824} C_VEL
LIN {X 0,Y 265.571,Z 900.667,A -85,B 0,C 180,E1 20912.374,E2 20912.374} C_VEL
LIN {X 0,Y 260.629,Z 908.618,A -85,B 0,C 180,E1 20913.549,E2 20913.549} C_VEL
LIN {X 0,Y 250.229,Z 921.464,A -85,B 0,C 180,E1 20914.909,E2 20914.909} C_VEL
LIN {X 0,Y 239.468,Z 933.495,A -85,B 0,C 180,E1 20916.462,E2 20916.462} C_VEL
LIN {X 0,Y 219.161,Z 956.819,A -85,B 0,C 180,E1 20922.997,E2 20922.997} C_VEL
LIN {X 0,Y 200.456,Z 975.284,A -85,B 0,C 180,E1 20931.458,E2 20931.458} C_VEL
LIN {X 0,Y 185.448,Z 988.709,A -85,B 0,C 180,E1 20942.003,E2 20942.003} C_VEL
LIN {X 0,Y 175.628,Z 997.246,A -85,B 0,C 180,E1 20955.013,E2 20955.013} C_VEL
LIN {X 0,Y 172.829,Z 999.938,A -85,B 0,C 180,E1 20964.975,E2 20964.975} C_VEL
LIN {X 0,Y 172.865,Z 999.905,A -85,B 0,C 180,E1 20975.025,E2 20975.025} C_VEL
LIN {X 0,Y 176.921,Z 996.101,A -85,B 0,C 180,E1 20987.429,E2 20987.429} C_VEL
LIN {X 0,Y 186.779,Z 987.514,A -85,B 0,C 180,E1 20999.101,E2 20999.101} C_VEL
LIN {X 0,Y 202.416,Z 973.372,A -85,B 0,C 180,E1 21009.477,E2 21009.477} C_VEL
LIN {X 0,Y 221.886,Z 953.719,A -85,B 0,C 180,E1 21017.904,E2 21017.904} C_VEL
LIN {X 0,Y 242.355,Z 929.463,A -85,B 0,C 180,E1 21024.303,E2 21024.303} C_VEL
LIN {X 0,Y 259.696,Z 904.856,A -85,B 0,C 180,E1 21028.558,E2 21028.558} C_VEL
LIN {X 0,Y 261.878,Z 893.394,A -85,B 0,C 180,E1 21032.97,E2 21032.97} C_VEL
LIN {X 0,Y 262.922,Z 879.856,A -85,B 0,C 180,E1 21039.799,E2 21039.799} C_VEL
LIN {X 0,Y 263.238,Z 870.847,A -85,B 0,C 180,E1 21046.71,E2 21046.71} C_VEL
LIN {X 0,Y 264.38,Z 866.144,A -85,B 0,C 180,E1 21053.433,E2 21053.433} C_VEL
LIN {X 0,Y 265.067,Z 865.825,A -85,B 0,C 180,E1 21056.734,E2 21056.734} C_VEL
LIN {X 0,Y 266.561,Z 872.993,A -85,B 0,C 180,E1 21064.895,E2 21064.895} C_VEL
LIN {X 0,Y 268.599,Z 884.038,A -85,B 0,C 180,E1 21071.386,E2 21071.386} C_VEL
LIN {X 0,Y 270.309,Z 899.83,A -85,B 0,C 180,E1 21077.569,E2 21077.569} C_VEL
LIN {X 0,Y 269.932,Z 903.854,A -85,B 0,C 180,E1 21078.602,E2 21078.602} C_VEL
LIN {X 0,Y 249.15,Z 940.345,A -85,B 0,C 180,E1 21082.648,E2 21082.648} C_VEL
LIN {X 0,Y 227.671,Z 972.058,A -85,B 0,C 180,E1 21088.183,E2 21088.183} C_VEL
LIN {X 0,Y 205.957,Z 1000.617,A -85,B 0,C 180,E1 21096.039,E2 21096.039} C_VEL
LIN {X 0,Y 188.644,Z 1022.836,A -85,B 0,C 180,E1 21105.651,E2 21105.651} C_VEL
LIN {X 0,Y 176.361,Z 1040.487,A -85,B 0,C 180,E1 21117.551,E2 21117.551} C_VEL
LIN {X 0,Y 171.098,Z 1051.56,A -85,B 0,C 180,E1 21129.271,E2 21129.271} C_VEL
LIN {X 0,Y 170.234,Z 1057.579,A -85,B 0,C 180,E1 21139.754,E2 21139.754} C_VEL
LIN {X 0,Y 171.203,Z 1059.817,A -85,B 0,C 180,E1 21150,E2 21150} C_VEL
LIN {X 0,Y 170.225,Z 1057.592,A -85,B 0,C 180,E1 21160.246,E2 21160.246} C_VEL
LIN {X 0,Y 171.582,Z 1050.116,A -85,B 0,C 180,E1 21172.651,E2 21172.651} C_VEL
LIN {X 0,Y 179.376,Z 1035.758,A -85,B 0,C 180,E1 21186.215,E2 21186.215} C_VEL
LIN {X 0,Y 195.002,Z 1014.687,A -85,B 0,C 180,E1 21198.432,E2 21198.432} C_VEL
LIN {X 0,Y 216.135,Z 987.737,A -85,B 0,C 180,E1 21207.981,E2 21207.981} C_VEL
LIN {X 0,Y 238.026,Z 957.499,A -85,B 0,C 180,E1 21214.688,E2 21214.688} C_VEL
LIN {X 0,Y 258.868,Z 924.463,A -85,B 0,C 180,E1 21219.351,E2 21219.351} C_VEL
LIN {X 0,Y 270.321,Z 903.484,A -85,B 0,C 180,E1 21221.429,E2 21221.429} C_VEL
LIN {X 0,Y 269.542,Z 889.54,A -85,B 0,C 180,E1 21226.269,E2 21226.269} C_VEL
LIN {X 0,Y 267.639,Z 878.018,A -85,B 0,C 180,E1 21231.862,E2 21231.862} C_VEL
LIN {X 0,Y 265.806,Z 869.667,A -85,B 0,C 180,E1 21238.36,E2 21238.36} C_VEL
LIN {X 0,Y 265.297,Z 865.882,A -85,B 0,C 180,E1 21243.263,E2 21243.263} C_VEL
LIN {X 0,Y 263.846,Z 867.732,A -85,B 0,C 180,E1 21248.632,E2 21248.632} C_VEL
LIN {X 0,Y 263.301,Z 873.923,A -85,B 0,C 180,E1 21255.89,E2 21255.89} C_VEL
LIN {X 0,Y 262.778,Z 884.814,A -85,B 0,C 180,E1 21262.805,E2 21262.805} C_VEL
LIN {X 0,Y 261.375,Z 898.621,A -85,B 0,C 180,E1 21269.066,E2 21269.066} C_VEL
LIN {X 0,Y 259.962,Z 904.686,A -85,B 0,C 180,E1 21271.297,E2 21271.297} C_VEL
LIN {X 0,Y 239.468,Z 933.495,A -85,B 0,C 180,E1 21276.462,E2 21276.462} C_VEL
LIN {X 0,Y 228.29,Z 944.763,A -85,B 0,C 180,E1 21278.294,E2 21278.294} C_VEL
LIN {X 0,Y 216.877,Z 955.118,A -85,B 0,C 180,E1 21280.436,E2 21280.436} C_VEL
LIN {X 0,Y 196.325,Z 974.955,A -85,B 0,C 180,E1 21289.044,E2 21289.044} C_VEL
LIN {X 0,Y 179.908,Z 989.02,A -85,B 0,C 180,E1 21299.674,E2 21299.674} C_VEL
LIN {X 0,Y 169.452,Z 997.538,A -85,B 0,C 180,E1 21311.778,E2 21311.778} C_VEL
LIN {X 0,Y 165.071,Z 1001.287,A -85,B 0,C 180,E1 21324.738,E2 21324.738} C_VEL
LIN {X 0,Y 165.102,Z 1001.256,A -85,B 0,C 180,E1 21335.262,E2 21335.262} C_VEL
LIN {X 0,Y 169.484,Z 997.457,A -85,B 0,C 180,E1 21348.22,E2 21348.22} C_VEL
LIN {X 0,Y 181.378,Z 987.676,A -85,B 0,C 180,E1 21361.446,E2 21361.446} C_VEL
LIN {X 0,Y 198.378,Z 972.964,A -85,B 0,C 180,E1 21371.897,E2 21371.897} C_VEL
LIN {X 0,Y 217.916,Z 953.874,A -85,B 0,C 180,E1 21379.839,E2 21379.839} C_VEL
LIN {X 0,Y 239.224,Z 929.251,A -85,B 0,C 180,E1 21386.166,E2 21386.166} C_VEL
LIN {X 0,Y 255.025,Z 907.384,A -85,B 0,C 180,E1 21389.95,E2 21389.95} C_VEL
LIN {X 0,Y 257.42,Z 894.266,A -85,B 0,C 180,E1 21395.7,E2 21395.7} C_VEL
LIN {X 0,Y 258.67,Z 883.153,A -85,B 0,C 180,E1 21402.201,E2 21402.201} C_VEL
LIN {X 0,Y 259.293,Z 876.971,A -85,B 0,C 180,E1 21407.652,E2 21407.652} C_VEL
LIN {X 0,Y 260.495,Z 873.195,A -85,B 0,C 180,E1 21413.334,E2 21413.334} C_VEL
LIN {X 0,Y 261.315,Z 872.802,A -85,B 0,C 180,E1 21416.688,E2 21416.688} C_VEL
LIN {X 0,Y 262.449,Z 879.303,A -85,B 0,C 180,E1 21424.319,E2 21424.319} C_VEL
LIN {X 0,Y 264.112,Z 889.82,A -85,B 0,C 180,E1 21430.745,E2 21430.745} C_VEL
LIN {X 0,Y 265.24,Z 905.394,A -85,B 0,C 180,E1 21437.041,E2 21437.041} C_VEL
LIN {X 0,Y 252.158,Z 928.977,A -85,B 0,C 180,E1 21439.626,E2 21439.626} C_VEL
LIN {X 0,Y 230.748,Z 961.115,A -85,B 0,C 180,E1 21444.421,E2 21444.421} C_VEL
LIN {X 0,Y 208.21,Z 990.419,A -85,B 0,C 180,E1 21451.307,E2 21451.307} C_VEL
LIN {X 0,Y 187.993,Z 1014.881,A -85,B 0,C 180,E1 21460.5,E2 21460.5} C_VEL
LIN {X 0,Y 172.644,Z 1034.239,A -85,B 0,C 180,E1 21472.131,E2 21472.131} C_VEL
LIN {X 0,Y 164.271,Z 1048.085,A -85,B 0,C 180,E1 21485.458,E2 21485.458} C_VEL
LIN {X 0,Y 162.388,Z 1055.448,A -85,B 0,C 180,E1 21497.501,E2 21497.501} C_VEL
LIN {X 0,Y 162.64,Z 1057.801,A -85,B 0,C 180,E1 21504.658,E2 21504.658} C_VEL
LIN {X 0,Y 163.405,Z 1058.466,A -85,B 0,C 180,E1 21510,E2 21510} C_VEL
LIN {X 0,Y 162.409,Z 1056.214,A -85,B 0,C 180,E1 21520.745,E2 21520.745} C_VEL
LIN {X 0,Y 163.59,Z 1049.809,A -85,B 0,C 180,E1 21532.234,E2 21532.234} C_VEL
LIN {X 0,Y 170.406,Z 1037.529,A -85,B 0,C 180,E1 21545.274,E2 21545.274} C_VEL
LIN {X 0,Y 184.68,Z 1018.925,A -85,B 0,C 180,E1 21557.545,E2 21557.545} C_VEL
LIN {X 0,Y 204.59,Z 994.982,A -85,B 0,C 180,E1 21567.326,E2 21567.326} C_VEL
LIN {X 0,Y 226.67,Z 966.825,A -85,B 0,C 180,E1 21574.508,E2 21574.508} C_VEL
LIN {X 0,Y 249.099,Z 934.131,A -85,B 0,C 180,E1 21579.762,E2 21579.762} C_VEL
LIN {X 0,Y 265.353,Z 906.058,A -85,B 0,C 180,E1 21582.776,E2 21582.776} C_VEL
LIN {X 0,Y 264.426,Z 891.678,A -85,B 0,C 180,E1 21588.432,E2 21588.432} C_VEL
LIN {X 0,Y 262.973,Z 881.714,A -85,B 0,C 180,E1 21594.04,E2 21594.04} C_VEL
LIN {X 0,Y 261.586,Z 873.912,A -85,B 0,C 180,E1 21601.65,E2 21601.65} C_VEL
LIN {X 0,Y 261.536,Z 872.87,A -85,B 0,C 180,E1 21603.31,E2 21603.31} C_VEL
LIN {X 0,Y 260.083,Z 874.496,A -85,B 0,C 180,E1 21608.272,E2 21608.272} C_VEL
LIN {X 0,Y 259.097,Z 880.06,A -85,B 0,C 180,E1 21615.235,E2 21615.235} C_VEL
LIN {X 0,Y 258.125,Z 890.012,A -85,B 0,C 180,E1 21621.911,E2 21621.911} C_VEL
LIN {X 0,Y 256.102,Z 903.149,A -85,B 0,C 180,E1 21628.212,E2 21628.212} C_VEL
LIN {X 0,Y 254.477,Z 908.621,A -85,B 0,C 180,E1 21630.162,E2 21630.162} C_VEL
LIN {X 0,Y 233.869,Z 936.193,A -85,B 0,C 180,E1 21635.228,E2 21635.228} C_VEL
LIN {X 0,Y 216.877,Z 955.118,A -85,B 0,C 180,E1 21640.436,E2 21640.436} C_VEL
LIN {X 0,Y 205.4,Z 964.72,A -85,B 0,C 180,E1 21642.932,E2 21642.932} C_VEL
LIN {X 0,Y 194,Z 973.28,A -85,B 0,C 180,E1 21645.851,E2 21645.851} C_VEL
LIN {X 0,Y 176.191,Z 987.987,A -85,B 0,C 180,E1 21656.046,E2 21656.046} C_VEL
LIN {X 0,Y 163.739,Z 997.539,A -85,B 0,C 180,E1 21668.294,E2 21668.294} C_VEL
LIN {X 0,Y 158.435,Z 1001.645,A -85,B 0,C 180,E1 21678.982,E2 21678.982} C_VEL
LIN {X 0,Y 157.287,Z 1002.918,A -85,B 0,C 180,E1 21690,E2 21690} C_VEL
LIN {X 0,Y 158.454,Z 1001.598,A -85,B 0,C 180,E1 21701.017,E2 21701.017} C_VEL
LIN {X 0,Y 166.182,Z 995.629,A -85,B 0,C 180,E1 21714.754,E2 21714.754} C_VEL
LIN {X 0,Y 179.505,Z 985.274,A -85,B 0,C 180,E1 21726.186,E2 21726.186} C_VEL
LIN {X 0,Y 198.731,Z 968.933,A -85,B 0,C 180,E1 21736.142,E2 21736.142} C_VEL
LIN {X 0,Y 219.198,Z 948.797,A -85,B 0,C 180,E1 21743.411,E2 21743.411} C_VEL
LIN {X 0,Y 240.548,Z 923.694,A -85,B 0,C 180,E1 21749.043,E2 21749.043} C_VEL
LIN {X 0,Y 249.804,Z 911.053,A -85,B 0,C 180,E1 21751.113,E2 21751.113} C_VEL
LIN {X 0,Y 252.696,Z 898.265,A -85,B 0,C 180,E1 21757.092,E2 21757.092} C_VEL
LIN {X 0,Y 254.155,Z 889.247,A -85,B 0,C 180,E1 21762.682,E2 21762.682} C_VEL
LIN {X 0,Y 255.478,Z 882.218,A -85,B 0,C 180,E1 21769.769,E2 21769.769} C_VEL
LIN {X 0,Y 256.5,Z 880.179,A -85,B 0,C 180,E1 21773.23,E2 21773.23} C_VEL
LIN {X 0,Y 257.474,Z 879.709,A -85,B 0,C 180,E1 21776.638,E2 21776.638} C_VEL
LIN {X 0,Y 258.401,Z 886.467,A -85,B 0,C 180,E1 21784.463,E2 21784.463} C_VEL
LIN {X 0,Y 259.64,Z 897.219,A -85,B 0,C 180,E1 21790.932,E2 21790.932} C_VEL
LIN {X 0,Y 260.055,Z 909.45,A -85,B 0,C 180,E1 21796.003,E2 21796.003} C_VEL
LIN {X 0,Y 238.215,Z 944.418,A -85,B 0,C 180,E1 21800.029,E2 21800.029} C_VEL
LIN {X 0,Y 214.54,Z 976.038,A -85,B 0,C 180,E1 21805.874,E2 21805.874} C_VEL
LIN {X 0,Y 190.405,Z 1004.563,A -85,B 0,C 180,E1 21814.609,E2 21814.609} C_VEL
LIN {X 0,Y 170.411,Z 1027.447,A -85,B 0,C 180,E1 21826.485,E2 21826.485} C_VEL
LIN {X 0,Y 158.768,Z 1043.156,A -85,B 0,C 180,E1 21840.038,E2 21840.038} C_VEL
LIN {X 0,Y 154.811,Z 1052.228,A -85,B 0,C 180,E1 21852.939,E2 21852.939} C_VEL
LIN {X 0,Y 154.8,Z 1056.436,A -85,B 0,C 180,E1 21864.387,E2 21864.387} C_VEL
LIN {X 0,Y 155.61,Z 1057.116,A -85,B 0,C 180,E1 21870,E2 21870} C_VEL
LIN {X 0,Y 154.556,Z 1054.726,A -85,B 0,C 180,E1 21881.551,E2 21881.551} C_VEL
LIN {X 0,Y 156.8,Z 1046.711,A -85,B 0,C 180,E1 21895.753,E2 21895.753} C_VEL
LIN {X 0,Y 167.442,Z 1031.149,A -85,B 0,C 180,E1 21910.96,E2 21910.96} C_VEL
LIN {X 0,Y 185.581,Z 1010.162,A -85,B 0,C 180,E1 21923.05,E2 21923.05} C_VEL
LIN {X 0,Y 207.847,Z 984.439,A -85,B 0,C 180,E1 21931.999,E2 21931.999} C_VEL
LIN {X 0,Y 231.4,Z 954.247,A -85,B 0,C 180,E1 21938.458,E2 21938.458} C_VEL
LIN {X 0,Y 253.499,Z 921.082,A -85,B 0,C 180,E1 21942.858,E2 21942.858} C_VEL
LIN {X 0,Y 260.167,Z 909.591,A -85,B 0,C 180,E1 21943.994,E2 21943.994} C_VEL
LIN {X 0,Y 259.644,Z 895.591,A -85,B 0,C 180,E1 21949.917,E2 21949.917} C_VEL
LIN {X 0,Y 258.298,Z 885.392,A -85,B 0,C 180,E1 21956.631,E2 21956.631} C_VEL
LIN {X 0,Y 257.681,Z 879.8,A -85,B 0,C 180,E1 21963.359,E2 21963.359} C_VEL
LIN {X 0,Y 255.559,Z 882.549,A -85,B 0,C 180,E1 21970.228,E2 21970.228} C_VEL
LIN {X 0,Y 254.572,Z 887.893,A -85,B 0,C 180,E1 21976.102,E2 21976.102} C_VEL
LIN {X 0,Y 252.833,Z 898.514,A -85,B 0,C 180,E1 21982.895,E2 21982.895} C_VEL
LIN {X 0,Y 250.34,Z 910.037,A -85,B 0,C 180,E1 21988.361,E2 21988.361} C_VEL
LIN {X 0,Y 247.681,Z 914.281,A -85,B 0,C 180,E1 21989.263,E2 21989.263} C_VEL
LIN {X 0,Y 226.855,Z 940.569,A -85,B 0,C 180,E1 21994.337,E2 21994.337} C_VEL
LIN {X 0,Y 205.68,Z 962.582,A -85,B 0,C 180,E1 22001.019,E2 22001.019} C_VEL
LIN {X 0,Y 194,Z 973.28,A -85,B 0,C 180,E1 22005.851,E2 22005.851} C_VEL
LIN {X 0,Y 182.668,Z 981.014,A -85,B 0,C 180,E1 22009.201,E2 22009.201} C_VEL
LIN {X 0,Y 171.9,Z 987.77,A -85,B 0,C 180,E1 22013.08,E2 22013.08} C_VEL
LIN {X 0,Y 158.043,Z 997.853,A -85,B 0,C 180,E1 22025.255,E2 22025.255} C_VEL
LIN {X 0,Y 150.786,Z 1002.994,A -85,B 0,C 180,E1 22038.416,E2 22038.416} C_VEL
LIN {X 0,Y 149.497,Z 1004.268,A -85,B 0,C 180,E1 22050,E2 22050} C_VEL
LIN {X 0,Y 150.803,Z 1002.95,A -85,B 0,C 180,E1 22061.584,E2 22061.584} C_VEL
LIN {X 0,Y 159.607,Z 996.635,A -85,B 0,C 180,E1 22076.466,E2 22076.466} C_VEL
LIN {X 0,Y 175.351,Z 985.011,A -85,B 0,C 180,E1 22089.034,E2 22089.034} C_VEL
LIN {X 0,Y 196.167,Z 967.908,A -85,B 0,C 180,E1 22098.906,E2 22098.906} C_VEL
LIN {X 0,Y 218.631,Z 946.098,A -85,B 0,C 180,E1 22106.2,E2 22106.2} C_VEL
LIN {X 0,Y 241.982,Z 918.285,A -85,B 0,C 180,E1 22111.809,E2 22111.809} C_VEL
LIN {X 0,Y 245.077,Z 913.485,A -85,B 0,C 180,E1 22112.838,E2 22112.838} C_VEL
LIN {X 0,Y 248.09,Z 902.321,A -85,B 0,C 180,E1 22118.533,E2 22118.533} C_VEL
LIN {X 0,Y 250.206,Z 892.561,A -85,B 0,C 180,E1 22125.503,E2 22125.503} C_VEL
LIN {X 0,Y 252.292,Z 887.055,A -85,B 0,C 180,E1 22133.116,E2 22133.116} C_VEL
LIN {X 0,Y 253.331,Z 886.46,A -85,B 0,C 180,E1 22136.583,E2 22136.583} C_VEL
LIN {X 0,Y 253.961,Z 892.061,A -85,B 0,C 180,E1 22143.426,E2 22143.426} C_VEL
LIN {X 0,Y 254.753,Z 901.128,A -85,B 0,C 180,E1 22149.414,E2 22149.414} C_VEL
LIN {X 0,Y 254.942,Z 912.714,A -85,B 0,C 180,E1 22154.614,E2 22154.614} C_VEL
LIN {X 0,Y 231.544,Z 948.314,A -85,B 0,C 180,E1 22158.926,E2 22158.926} C_VEL
LIN {X 0,Y 206.735,Z 979.455,A -85,B 0,C 180,E1 22165.005,E2 22165.005} C_VEL
LIN {X 0,Y 183.955,Z 1004.915,A -85,B 0,C 180,E1 22173.227,E2 22173.227} C_VEL
LIN {X 0,Y 164.384,Z 1025.97,A -85,B 0,C 180,E1 22184.456,E2 22184.456} C_VEL
LIN {X 0,Y 151.6,Z 1041.708,A -85,B 0,C 180,E1 22198.464,E2 22198.464} C_VEL
LIN {X 0,Y 147.064,Z 1050.818,A -85,B 0,C 180,E1 22212.01,E2 22212.01} C_VEL
LIN {X 0,Y 146.936,Z 1055.066,A -85,B 0,C 180,E1 22224.085,E2 22224.085} C_VEL
LIN {X 0,Y 147.804,Z 1055.764,A -85,B 0,C 180,E1 22230,E2 22230} C_VEL
LIN {X 0,Y 146.709,Z 1053.44,A -85,B 0,C 180,E1 22241.911,E2 22241.911} C_VEL
LIN {X 0,Y 148.838,Z 1046.302,A -85,B 0,C 180,E1 22255.614,E2 22255.614} C_VEL
LIN {X 0,Y 157.992,Z 1033.31,A -85,B 0,C 180,E1 22269.932,E2 22269.932} C_VEL
LIN {X 0,Y 174.901,Z 1014.657,A -85,B 0,C 180,E1 22282.324,E2 22282.324} C_VEL
LIN {X 0,Y 197.513,Z 990.268,A -85,B 0,C 180,E1 22291.986,E2 22291.986} C_VEL
LIN {X 0,Y 221.263,Z 961.993,A -85,B 0,C 180,E1 22298.794,E2 22298.794} C_VEL
LIN {X 0,Y 244.187,Z 930.291,A -85,B 0,C 180,E1 22303.503,E2 22303.503} C_VEL
LIN {X 0,Y 255.074,Z 912.842,A -85,B 0,C 180,E1 22305.377,E2 22305.377} C_VEL
LIN {X 0,Y 254.834,Z 899.655,A -85,B 0,C 180,E1 22311.45,E2 22311.45} C_VEL
LIN {X 0,Y 253.778,Z 890.558,A -85,B 0,C 180,E1 22318.272,E2 22318.272} C_VEL
LIN {X 0,Y 253.521,Z 886.576,A -85,B 0,C 180,E1 22323.414,E2 22323.414} C_VEL
LIN {X 0,Y 251.247,Z 889.444,A -85,B 0,C 180,E1 22330.405,E2 22330.405} C_VEL
LIN {X 0,Y 249.808,Z 895.424,A -85,B 0,C 180,E1 22336.719,E2 22336.719} C_VEL
LIN {X 0,Y 247.322,Z 905.97,A -85,B 0,C 180,E1 22343.332,E2 22343.332} C_VEL
LIN {X 0,Y 245.022,Z 914.253,A -85,B 0,C 180,E1 22347.391,E2 22347.391} C_VEL
LIN {X 0,Y 223.412,Z 941.054,A -85,B 0,C 180,E1 22352.468,E2 22352.468} C_VEL
LIN {X 0,Y 201.845,Z 962.847,A -85,B 0,C 180,E1 22358.904,E2 22358.904} C_VEL
LIN {X 0,Y 180.673,Z 980.953,A -85,B 0,C 180,E1 22367.904,E2 22367.904} C_VEL
LIN {X 0,Y 171.9,Z 987.77,A -85,B 0,C 180,E1 22373.08,E2 22373.08} C_VEL
LIN {X 0,Y 161.699,Z 993.558,A -85,B 0,C 180,E1 22377.556,E2 22377.556} C_VEL
LIN {X 0,Y 152.18,Z 998.367,A -85,B 0,C 180,E1 22382.657,E2 22382.657} C_VEL
LIN {X 0,Y 143.16,Z 1004.345,A -85,B 0,C 180,E1 22397.79,E2 22397.79} C_VEL
LIN {X 0,Y 141.733,Z 1005.612,A -85,B 0,C 180,E1 22410,E2 22410} C_VEL
LIN {X 0,Y 143.177,Z 1004.299,A -85,B 0,C 180,E1 22422.21,E2 22422.21} C_VEL
LIN {X 0,Y 151.414,Z 998.836,A -85,B 0,C 180,E1 22436.421,E2 22436.421} C_VEL
LIN {X 0,Y 167.114,Z 988.007,A -85,B 0,C 180,E1 22449.359,E2 22449.359} C_VEL
LIN {X 0,Y 187.584,Z 972.257,A -85,B 0,C 180,E1 22459.302,E2 22459.302} C_VEL
LIN {X 0,Y 210.259,Z 951.647,A -85,B 0,C 180,E1 22466.8,E2 22466.8} C_VEL
LIN {X 0,Y 232.943,Z 926.619,A -85,B 0,C 180,E1 22472.319,E2 22472.319} C_VEL
LIN {X 0,Y 239.804,Z 917.846,A -85,B 0,C 180,E1 22473.785,E2 22473.785} C_VEL
LIN {X 0,Y 243.489,Z 906.351,A -85,B 0,C 180,E1 22480.045,E2 22480.045} C_VEL
LIN {X 0,Y 245.597,Z 898.949,A -85,B 0,C 180,E1 22485.735,E2 22485.735} C_VEL
LIN {X 0,Y 247.872,Z 893.811,A -85,B 0,C 180,E1 22492.993,E2 22492.993} C_VEL
LIN {X 0,Y 249.075,Z 893.173,A -85,B 0,C 180,E1 22496.525,E2 22496.525} C_VEL
LIN {X 0,Y 249.603,Z 899.941,A -85,B 0,C 180,E1 22504.357,E2 22504.357} C_VEL
LIN {X 0,Y 250.005,Z 910.001,A -85,B 0,C 180,E1 22510.476,E2 22510.476} C_VEL
LIN {X 0,Y 249.762,Z 916.033,A -85,B 0,C 180,E1 22513.229,E2 22513.229} C_VEL
LIN {X 0,Y 226.698,Z 949.658,A -85,B 0,C 180,E1 22517.385,E2 22517.385} C_VEL
LIN {X 0,Y 201.694,Z 979.726,A -85,B 0,C 180,E1 22523.303,E2 22523.303} C_VEL
LIN {X 0,Y 177.835,Z 1005.032,A -85,B 0,C 180,E1 22531.641,E2 22531.641} C_VEL
LIN {X 0,Y 157.846,Z 1025.241,A -85,B 0,C 180,E1 22542.819,E2 22542.819} C_VEL
LIN {X 0,Y 144.308,Z 1040.541,A -85,B 0,C 180,E1 22557.089,E2 22557.089} C_VEL
LIN {X 0,Y 139.33,Z 1049.404,A -85,B 0,C 180,E1 22570.974,E2 22570.974} C_VEL
LIN {X 0,Y 139.086,Z 1053.698,A -85,B 0,C 180,E1 22583.75,E2 22583.75} C_VEL
LIN {X 0,Y 139.974,Z 1054.407,A -85,B 0,C 180,E1 22590,E2 22590} C_VEL
LIN {X 0,Y 138.857,Z 1052.047,A -85,B 0,C 180,E1 22602.595,E2 22602.595} C_VEL
LIN {X 0,Y 141.405,Z 1044.867,A -85,B 0,C 180,E1 22617.067,E2 22617.067} C_VEL
LIN {X 0,Y 152.401,Z 1031.026,A -85,B 0,C 180,E1 22632.689,E2 22632.689} C_VEL
LIN {X 0,Y 171.15,Z 1011.877,A -85,B 0,C 180,E1 22645.238,E2 22645.238} C_VEL
LIN {X 0,Y 194.385,Z 987.97,A -85,B 0,C 180,E1 22654.442,E2 22654.442} C_VEL
LIN {X 0,Y 218.361,Z 960.426,A -85,B 0,C 180,E1 22660.852,E2 22660.852} C_VEL
LIN {X 0,Y 242.195,Z 928.32,A -85,B 0,C 180,E1 22665.419,E2 22665.419} C_VEL
LIN {X 0,Y 249.882,Z 916.238,A -85,B 0,C 180,E1 22666.734,E2 22666.734} C_VEL
LIN {X 0,Y 250.036,Z 905.203,A -85,B 0,C 180,E1 22672.161,E2 22672.161} C_VEL
LIN {X 0,Y 249.42,Z 897.29,A -85,B 0,C 180,E1 22678.252,E2 22678.252} C_VEL
LIN {X 0,Y 249.258,Z 893.29,A -85,B 0,C 180,E1 22683.473,E2 22683.473} C_VEL
LIN {X 0,Y 246.641,Z 896.398,A -85,B 0,C 180,E1 22690.843,E2 22690.843} C_VEL
LIN {X 0,Y 244.763,Z 902.452,A -85,B 0,C 180,E1 22697.075,E2 22697.075} C_VEL
LIN {X 0,Y 241.443,Z 913.623,A -85,B 0,C 180,E1 22703.935,E2 22703.935} C_VEL
LIN {X 0,Y 239.312,Z 918.825,A -85,B 0,C 180,E1 22706.273,E2 22706.273} C_VEL
LIN {X 0,Y 215.697,Z 946.399,A -85,B 0,C 180,E1 22711.68,E2 22711.68} C_VEL
LIN {X 0,Y 191.954,Z 968.719,A -85,B 0,C 180,E1 22718.927,E2 22718.927} C_VEL
LIN {X 0,Y 170.885,Z 985.386,A -85,B 0,C 180,E1 22728.358,E2 22728.358} C_VEL
LIN {X 0,Y 154.171,Z 997.069,A -85,B 0,C 180,E1 22740.593,E2 22740.593} C_VEL
LIN {X 0,Y 152.18,Z 998.367,A -85,B 0,C 180,E1 22742.657,E2 22742.657} C_VEL
LIN {X 0,Y 143.669,Z 1002.304,A -85,B 0,C 180,E1 22748.406,E2 22748.406} C_VEL
LIN {X 0,Y 136.338,Z 1005.095,A -85,B 0,C 180,E1 22754.846,E2 22754.846} C_VEL
LIN {X 0,Y 133.943,Z 1006.962,A -85,B 0,C 180,E1 22770,E2 22770} C_VEL
LIN {X 0,Y 135.577,Z 1005.649,A -85,B 0,C 180,E1 22782.906,E2 22782.906} C_VEL
LIN {X 0,Y 144.722,Z 1000.021,A -85,B 0,C 180,E1 22798.084,E2 22798.084} C_VEL
LIN {X 0,Y 162.027,Z 988.745,A -85,B 0,C 180,E1 22811.65,E2 22811.65} C_VEL
LIN {X 0,Y 184.837,Z 971.804,A -85,B 0,C 180,E1 22822.008,E2 22822.008} C_VEL
LIN {X 0,Y 208.944,Z 950.281,A -85,B 0,C 180,E1 22829.357,E2 22829.357} C_VEL
LIN {X 0,Y 232.447,Z 924.446,A -85,B 0,C 180,E1 22834.652,E2 22834.652} C_VEL
LIN {X 0,Y 235.441,Z 920.032,A -85,B 0,C 180,E1 22835.855,E2 22835.855} C_VEL
LIN {X 0,Y 239.031,Z 910.183,A -85,B 0,C 180,E1 22841.821,E2 22841.821} C_VEL
LIN {X 0,Y 241.27,Z 904.004,A -85,B 0,C 180,E1 22847.323,E2 22847.323} C_VEL
LIN {X 0,Y 243.656,Z 900.208,A -85,B 0,C 180,E1 22853.819,E2 22853.819} C_VEL
LIN {X 0,Y 244.616,Z 899.742,A -85,B 0,C 180,E1 22856.461,E2 22856.461} C_VEL
LIN {X 0,Y 244.953,Z 905.62,A -85,B 0,C 180,E1 22863.553,E2 22863.553} C_VEL
LIN {X 0,Y 244.911,Z 914.992,A -85,B 0,C 180,E1 22869.639,E2 22869.639} C_VEL
LIN {X 0,Y 244.627,Z 919.748,A -85,B 0,C 180,E1 22871.919,E2 22871.919} C_VEL
LIN {X 0,Y 218.952,Z 954.874,A -85,B 0,C 180,E1 22876.378,E2 22876.378} C_VEL
LIN {X 0,Y 192.548,Z 984.543,A -85,B 0,C 180,E1 22882.719,E2 22882.719} C_VEL
LIN {X 0,Y 167.341,Z 1009.521,A -85,B 0,C 180,E1 22891.984,E2 22891.984} C_VEL
LIN {X 0,Y 146.423,Z 1029.423,A -85,B 0,C 180,E1 22905.007,E2 22905.007} C_VEL
LIN {X 0,Y 134.099,Z 1043.403,A -85,B 0,C 180,E1 22921.325,E2 22921.325} C_VEL
LIN {X 0,Y 131.052,Z 1050.642,A -85,B 0,C 180,E1 22936.641,E2 22936.641} C_VEL
LIN {X 0,Y 132.137,Z 1053.05,A -85,B 0,C 180,E1 22950,E2 22950} C_VEL
LIN {X 0,Y 131.019,Z 1050.654,A -85,B 0,C 180,E1 22963.362,E2 22963.362} C_VEL
LIN {X 0,Y 134.855,Z 1042.409,A -85,B 0,C 180,E1 22980.344,E2 22980.344} C_VEL
LIN {X 0,Y 148.925,Z 1027.052,A -85,B 0,C 180,E1 22997.092,E2 22997.092} C_VEL
LIN {X 0,Y 171.025,Z 1006.11,A -85,B 0,C 180,E1 23009.667,E2 23009.667} C_VEL
LIN {X 0,Y 197.04,Z 979.964,A -85,B 0,C 180,E1 23018.514,E2 23018.514} C_VEL
LIN {X 0,Y 223.16,Z 949.787,A -85,B 0,C 180,E1 23024.423,E2 23024.423} C_VEL
LIN {X 0,Y 244.78,Z 919.807,A -85,B 0,C 180,E1 23028.096,E2 23028.096} C_VEL
LIN {X 0,Y 245.17,Z 909.305,A -85,B 0,C 180,E1 23033.787,E2 23033.787} C_VEL
LIN {X 0,Y 244.792,Z 902.349,A -85,B 0,C 180,E1 23039.991,E2 23039.991} C_VEL
LIN {X 0,Y 244.791,Z 899.872,A -85,B 0,C 180,E1 23043.536,E2 23043.536} C_VEL
LIN {X 0,Y 241.974,Z 902.858,A -85,B 0,C 180,E1 23050.808,E2 23050.808} C_VEL
LIN {X 0,Y 240.06,Z 907.898,A -85,B 0,C 180,E1 23056.223,E2 23056.223} C_VEL
LIN {X 0,Y 236.58,Z 917.446,A -85,B 0,C 180,E1 23062.567,E2 23062.567} C_VEL
LIN {X 0,Y 235.157,Z 921.201,A -85,B 0,C 180,E1 23064.58,E2 23064.58} C_VEL
LIN {X 0,Y 210.305,Z 949.18,A -85,B 0,C 180,E1 23070.245,E2 23070.245} C_VEL
LIN {X 0,Y 185.769,Z 971.19,A -85,B 0,C 180,E1 23077.559,E2 23077.559} C_VEL
LIN {X 0,Y 162.821,Z 988.285,A -85,B 0,C 180,E1 23087.795,E2 23087.795} C_VEL
LIN {X 0,Y 147.424,Z 998.418,A -85,B 0,C 180,E1 23099.104,E2 23099.104} C_VEL
LIN {X 0,Y 136.338,Z 1005.095,A -85,B 0,C 180,E1 23114.846,E2 23114.846} C_VEL
LIN {X 0,Y 132.186,Z 1006.729,A -85,B 0,C 180,E1 23120.123,E2 23120.123} C_VEL
LIN {X 0,Y 126.161,Z 1008.255,A -85,B 0,C 180,E1 23128.494,E2 23128.494} C_VEL
LIN {X 0,Y 126.133,Z 1008.286,A -85,B 0,C 180,E1 23129.493,E2 23129.493} C_VEL
LIN {X 0,Y 127.991,Z 1007,A -85,B 0,C 180,E1 23143.685,E2 23143.685} C_VEL
LIN {X 0,Y 137.882,Z 1001.373,A -85,B 0,C 180,E1 23159.612,E2 23159.612} C_VEL
LIN {X 0,Y 155.333,Z 990.73,A -85,B 0,C 180,E1 23173.022,E2 23173.022} C_VEL
LIN {X 0,Y 178.556,Z 974.403,A -85,B 0,C 180,E1 23183.409,E2 23183.409} C_VEL
LIN {X 0,Y 203.818,Z 952.882,A -85,B 0,C 180,E1 23190.913,E2 23190.913} C_VEL
LIN {X 0,Y 228.114,Z 927.219,A -85,B 0,C 180,E1 23196.198,E2 23196.198} C_VEL
LIN {X 0,Y 230.336,Z 924.305,A -85,B 0,C 180,E1 23196.958,E2 23196.958} C_VEL
LIN {X 0,Y 234.476,Z 914.68,A -85,B 0,C 180,E1 23203.259,E2 23203.259} C_VEL
LIN {X 0,Y 236.993,Z 909.233,A -85,B 0,C 180,E1 23208.962,E2 23208.962} C_VEL
LIN {X 0,Y 238.524,Z 906.996,A -85,B 0,C 180,E1 23212.717,E2 23212.717} C_VEL
LIN {X 0,Y 239.985,Z 906.185,A -85,B 0,C 180,E1 23216.393,E2 23216.393} C_VEL
LIN {X 0,Y 240.101,Z 912.186,A -85,B 0,C 180,E1 23223.624,E2 23223.624} C_VEL
LIN {X 0,Y 239.652,Z 922.012,A -85,B 0,C 180,E1 23229.853,E2 23229.853} C_VEL
LIN {X 0,Y 238.523,Z 924.813,A -85,B 0,C 180,E1 23230.715,E2 23230.715} C_VEL
LIN {X 0,Y 213.433,Z 957.111,A -85,B 0,C 180,E1 23234.874,E2 23234.874} C_VEL
LIN {X 0,Y 186.835,Z 985.58,A -85,B 0,C 180,E1 23241.08,E2 23241.08} C_VEL
LIN {X 0,Y 160.459,Z 1010.265,A -85,B 0,C 180,E1 23250.573,E2 23250.573} C_VEL
LIN {X 0,Y 139.622,Z 1028.834,A -85,B 0,C 180,E1 23263.386,E2 23263.386} C_VEL
LIN {X 0,Y 127.597,Z 1041.175,A -85,B 0,C 180,E1 23278.17,E2 23278.17} C_VEL
LIN {X 0,Y 123.225,Z 1049.245,A -85,B 0,C 180,E1 23295.775,E2 23295.775} C_VEL
LIN {X 0,Y 124.299,Z 1051.692,A -85,B 0,C 180,E1 23310,E2 23310} C_VEL
LIN {X 0,Y 123.198,Z 1049.259,A -85,B 0,C 180,E1 23324.228,E2 23324.228} C_VEL
LIN {X 0,Y 127.565,Z 1041.205,A -85,B 0,C 180,E1 23341.831,E2 23341.831} C_VEL
LIN {X 0,Y 141.743,Z 1026.959,A -85,B 0,C 180,E1 23358.39,E2 23358.39} C_VEL
LIN {X 0,Y 165.595,Z 1005.846,A -85,B 0,C 180,E1 23371.64,E2 23371.64} C_VEL
LIN {X 0,Y 192.757,Z 979.86,A -85,B 0,C 180,E1 23380.48,E2 23380.48} C_VEL
LIN {X 0,Y 219.504,Z 950.13,A -85,B 0,C 180,E1 23386.235,E2 23386.235} C_VEL
LIN {X 0,Y 239.674,Z 923.281,A -85,B 0,C 180,E1 23389.546,E2 23389.546} C_VEL
LIN {X 0,Y 240.225,Z 913.469,A -85,B 0,C 180,E1 23395.473,E2 23395.473} C_VEL
LIN {X 0,Y 240.132,Z 907.389,A -85,B 0,C 180,E1 23401.797,E2 23401.797} C_VEL
LIN {X 0,Y 240.129,Z 906.343,A -85,B 0,C 180,E1 23403.605,E2 23403.605} C_VEL
LIN {X 0,Y 237.09,Z 909.467,A -85,B 0,C 180,E1 23411.034,E2 23411.034} C_VEL
LIN {X 0,Y 234.589,Z 914.92,A -85,B 0,C 180,E1 23416.761,E2 23416.761} C_VEL
LIN {X 0,Y 230.18,Z 924.953,A -85,B 0,C 180,E1 23423.231,E2 23423.231} C_VEL
LIN {X 0,Y 206.499,Z 950.577,A -85,B 0,C 180,E1 23428.382,E2 23428.382} C_VEL
LIN {X 0,Y 181.77,Z 972.06,A -85,B 0,C 180,E1 23435.385,E2 23435.385} C_VEL
LIN {X 0,Y 159.543,Z 988.101,A -85,B 0,C 180,E1 23444.626,E2 23444.626} C_VEL
LIN {X 0,Y 140.767,Z 999.774,A -85,B 0,C 180,E1 23457.469,E2 23457.469} C_VEL
LIN {X 0,Y 130.93,Z 1005.357,A -85,B 0,C 180,E1 23469.703,E2 23469.703} C_VEL
LIN {X 0,Y 126.133,Z 1008.286,A -85,B 0,C 180,E1 23489.493,E2 23489.493} C_VEL
LIN {X 0,Y 124.095,Z 1008.665,A -85,B 0,C 180,E1 23495.395,E2 23495.395} C_VEL
LIN {X 0,Y 120.533,Z 1008.325,A -85,B 0,C 180,E1 23504.584,E2 23504.584} C_VEL
LIN {X 0,Y 120.796,Z 1008.096,A -85,B 0,C 180,E1 23505.621,E2 23505.621} C_VEL
LIN {X 0,Y 131.146,Z 1002.728,A -85,B 0,C 180,E1 23521.299,E2 23521.299} C_VEL
LIN {X 0,Y 149.73,Z 992.09,A -85,B 0,C 180,E1 23535.057,E2 23535.057} C_VEL
LIN {X 0,Y 174.017,Z 975.781,A -85,B 0,C 180,E1 23545.472,E2 23545.472} C_VEL
LIN {X 0,Y 199.965,Z 954.463,A -85,B 0,C 180,E1 23552.815,E2 23552.815} C_VEL
LIN {X 0,Y 225.104,Z 928.682,A -85,B 0,C 180,E1 23558,E2 23558} C_VEL
LIN {X 0,Y 229.316,Z 920.367,A -85,B 0,C 180,E1 23563.716,E2 23563.716} C_VEL
LIN {X 0,Y 232.404,Z 914.771,A -85,B 0,C 180,E1 23570.094,E2 23570.094} C_VEL
LIN {X 0,Y 235.212,Z 912.576,A -85,B 0,C 180,E1 23576.319,E2 23576.319} C_VEL
LIN {X 0,Y 235.179,Z 917.641,A -85,B 0,C 180,E1 23582.777,E2 23582.777} C_VEL
LIN {X 0,Y 234.413,Z 926.579,A -85,B 0,C 180,E1 23588.885,E2 23588.885} C_VEL
LIN {X 0,Y 209.684,Z 957.53,A -85,B 0,C 180,E1 23592.998,E2 23592.998} C_VEL
LIN {X 0,Y 182.207,Z 985.739,A -85,B 0,C 180,E1 23599.096,E2 23599.096} C_VEL
LIN {X 0,Y 155.019,Z 1009.902,A -85,B 0,C 180,E1 23608.479,E2 23608.479} C_VEL
LIN {X 0,Y 132.654,Z 1028.492,A -85,B 0,C 180,E1 23621.838,E2 23621.838} C_VEL
LIN {X 0,Y 118.945,Z 1041.554,A -85,B 0,C 180,E1 23639.393,E2 23639.393} C_VEL
LIN {X 0,Y 115.419,Z 1047.846,A -85,B 0,C 180,E1 23654.79,E2 23654.79} C_VEL
LIN {X 0,Y 116.465,Z 1050.335,A -85,B 0,C 180,E1 23669.999,E2 23669.999} C_VEL
LIN {X 0,Y 115.392,Z 1047.861,A -85,B 0,C 180,E1 23685.212,E2 23685.212} C_VEL
LIN {X 0,Y 120.44,Z 1039.871,A -85,B 0,C 180,E1 23703.725,E2 23703.725} C_VEL
LIN {X 0,Y 136.289,Z 1025.495,A -85,B 0,C 180,E1 23721.041,E2 23721.041} C_VEL
LIN {X 0,Y 161.716,Z 1004.337,A -85,B 0,C 180,E1 23734.301,E2 23734.301} C_VEL
LIN {X 0,Y 190.101,Z 978.33,A -85,B 0,C 180,E1 23742.88,E2 23742.88} C_VEL
LIN {X 0,Y 217.402,Z 948.883,A -85,B 0,C 180,E1 23748.325,E2 23748.325} C_VEL
LIN {X 0,Y 234.536,Z 926.705,A -85,B 0,C 180,E1 23751.118,E2 23751.118} C_VEL
LIN {X 0,Y 235.266,Z 918.833,A -85,B 0,C 180,E1 23756.301,E2 23756.301} C_VEL
LIN {X 0,Y 235.353,Z 912.737,A -85,B 0,C 180,E1 23763.678,E2 23763.678} C_VEL
LIN {X 0,Y 231.793,Z 916.084,A -85,B 0,C 180,E1 23771.552,E2 23771.552} C_VEL
LIN {X 0,Y 228.725,Z 921.911,A -85,B 0,C 180,E1 23777.318,E2 23777.318} C_VEL
LIN {X 0,Y 225.042,Z 929.011,A -85,B 0,C 180,E1 23781.938,E2 23781.938} C_VEL
LIN {X 0,Y 199.396,Z 955.204,A -85,B 0,C 180,E1 23787.269,E2 23787.269} C_VEL
LIN {X 0,Y 173.339,Z 976.434,A -85,B 0,C 180,E1 23794.678,E2 23794.678} C_VEL
LIN {X 0,Y 148.537,Z 992.94,A -85,B 0,C 180,E1 23805.493,E2 23805.493} C_VEL
LIN {X 0,Y 131.094,Z 1002.826,A -85,B 0,C 180,E1 23818.689,E2 23818.689} C_VEL
LIN {X 0,Y 120.417,Z 1008.392,A -85,B 0,C 180,E1 23835.437,E2 23835.437} C_VEL
LIN {X 0,Y 118.4,Z 1009.654,A -85,B 0,C 180,E1 23850.001,E2 23850.001} C_VEL
LIN {X 0,Y 120.796,Z 1008.096,A -85,B 0,C 180,E1 23865.621,E2 23865.621} C_VEL
LIN {X 0,Y 121.018,Z 1006.839,A -85,B 0,C 180,E1 23873.901,E2 23873.901} C_VEL
LIN {X 0,Y 123.386,Z 1004.622,A -85,B 0,C 180,E1 23882.004,E2 23882.004} C_VEL
LIN {X 0,Y 144.305,Z 993.456,A -85,B 0,C 180,E1 23897.258,E2 23897.258} C_VEL
LIN {X 0,Y 169.939,Z 977.003,A -85,B 0,C 180,E1 23907.706,E2 23907.706} C_VEL
LIN {X 0,Y 196.535,Z 955.871,A -85,B 0,C 180,E1 23914.831,E2 23914.831} C_VEL
LIN {X 0,Y 220.307,Z 932.42,A -85,B 0,C 180,E1 23919.497,E2 23919.497} C_VEL
LIN {X 0,Y 224.779,Z 924.721,A -85,B 0,C 180,E1 23925.381,E2 23925.381} C_VEL
LIN {X 0,Y 228.422,Z 919.77,A -85,B 0,C 180,E1 23932.393,E2 23932.393} C_VEL
LIN {X 0,Y 230.166,Z 918.797,A -85,B 0,C 180,E1 23936.239,E2 23936.239} C_VEL
LIN {X 0,Y 230.024,Z 923.937,A -85,B 0,C 180,E1 23942.839,E2 23942.839} C_VEL
LIN {X 0,Y 229.12,Z 930.826,A -85,B 0,C 180,E1 23947.614,E2 23947.614} C_VEL
LIN {X 0,Y 201.173,Z 963.244,A -85,B 0,C 180,E1 23951.941,E2 23951.941} C_VEL
LIN {X 0,Y 171.777,Z 991.25,A -85,B 0,C 180,E1 23958.652,E2 23958.652} C_VEL
LIN {X 0,Y 143.782,Z 1014.15,A -85,B 0,C 180,E1 23968.877,E2 23968.877} C_VEL
LIN {X 0,Y 121.296,Z 1031.649,A -85,B 0,C 180,E1 23984.134,E2 23984.134} C_VEL
LIN {X 0,Y 109.492,Z 1042.897,A -85,B 0,C 180,E1 24003.28,E2 24003.28} C_VEL
LIN {X 0,Y 107.465,Z 1047.935,A -85,B 0,C 180,E1 24020.562,E2 24020.562} C_VEL
LIN {X 0,Y 108.614,Z 1048.975,A -85,B 0,C 180,E1 24029.999,E2 24029.999} C_VEL
LIN {X 0,Y 107.611,Z 1046.46,A -85,B 0,C 180,E1 24046.342,E2 24046.342} C_VEL
LIN {X 0,Y 113.066,Z 1038.914,A -85,B 0,C 180,E1 24065.142,E2 24065.142} C_VEL
LIN {X 0,Y 131.14,Z 1024.029,A -85,B 0,C 180,E1 24083.914,E2 24083.914} C_VEL
LIN {X 0,Y 157.909,Z 1003.106,A -85,B 0,C 180,E1 24096.957,E2 24096.957} C_VEL
LIN {X 0,Y 187.798,Z 976.812,A -85,B 0,C 180,E1 24105.332,E2 24105.332} C_VEL
LIN {X 0,Y 215.856,Z 947.298,A -85,B 0,C 180,E1 24110.512,E2 24110.512} C_VEL
LIN {X 0,Y 229.346,Z 930.805,A -85,B 0,C 180,E1 24112.404,E2 24112.404} C_VEL
LIN {X 0,Y 230.121,Z 923.428,A -85,B 0,C 180,E1 24117.842,E2 24117.842} C_VEL
LIN {X 0,Y 230.287,Z 918.964,A -85,B 0,C 180,E1 24123.759,E2 24123.759} C_VEL
LIN {X 0,Y 226.54,Z 922.28,A -85,B 0,C 180,E1 24131.555,E2 24131.555} C_VEL
LIN {X 0,Y 222.648,Z 928.75,A -85,B 0,C 180,E1 24137.827,E2 24137.827} C_VEL
LIN {X 0,Y 220.269,Z 932.718,A -85,B 0,C 180,E1 24140.435,E2 24140.435} C_VEL
LIN {X 0,Y 193.777,Z 958.552,A -85,B 0,C 180,E1 24145.732,E2 24145.732} C_VEL
LIN {X 0,Y 167.34,Z 979.032,A -85,B 0,C 180,E1 24153.078,E2 24153.078} C_VEL
LIN {X 0,Y 141.581,Z 995.108,A -85,B 0,C 180,E1 24164.12,E2 24164.12} C_VEL
LIN {X 0,Y 121.428,Z 1005.654,A -85,B 0,C 180,E1 24180.085,E2 24180.085} C_VEL
LIN {X 0,Y 112.886,Z 1009.743,A -85,B 0,C 180,E1 24194.441,E2 24194.441} C_VEL
LIN {X 0,Y 110.635,Z 1010.999,A -85,B 0,C 180,E1 24210.001,E2 24210.001} C_VEL
LIN {X 0,Y 113.186,Z 1009.518,A -85,B 0,C 180,E1 24226.365,E2 24226.365} C_VEL
LIN {X 0,Y 123.386,Z 1004.622,A -85,B 0,C 180,E1 24242.004,E2 24242.004} C_VEL
LIN {X 0,Y 127.659,Z 1001.648,A -85,B 0,C 180,E1 24249.656,E2 24249.656} C_VEL
LIN {X 0,Y 133.659,Z 997.718,A -85,B 0,C 180,E1 24256.692,E2 24256.692} C_VEL
LIN {X 0,Y 157.539,Z 983.908,A -85,B 0,C 180,E1 24267.236,E2 24267.236} C_VEL
LIN {X 0,Y 183.992,Z 965.027,A -85,B 0,C 180,E1 24274.843,E2 24274.843} C_VEL
LIN {X 0,Y 211.122,Z 940.701,A -85,B 0,C 180,E1 24280.318,E2 24280.318} C_VEL
LIN {X 0,Y 215.957,Z 935.657,A -85,B 0,C 180,E1 24281.413,E2 24281.413} C_VEL
LIN {X 0,Y 220.391,Z 929.089,A -85,B 0,C 180,E1 24287.221,E2 24287.221} C_VEL
LIN {X 0,Y 223.095,Z 925.92,A -85,B 0,C 180,E1 24292.334,E2 24292.334} C_VEL
LIN {X 0,Y 225.028,Z 924.942,A -85,B 0,C 180,E1 24296.153,E2 24296.153} C_VEL
LIN {X 0,Y 224.702,Z 930.161,A -85,B 0,C 180,E1 24302.906,E2 24302.906} C_VEL
LIN {X 0,Y 224.104,Z 933.983,A -85,B 0,C 180,E1 24305.826,E2 24305.826} C_VEL
LIN {X 0,Y 197.374,Z 963.936,A -85,B 0,C 180,E1 24309.963,E2 24309.963} C_VEL
LIN {X 0,Y 168.41,Z 990.427,A -85,B 0,C 180,E1 24316.132,E2 24316.132} C_VEL
LIN {X 0,Y 140.479,Z 1012.212,A -85,B 0,C 180,E1 24325.553,E2 24325.553} C_VEL
LIN {X 0,Y 116.043,Z 1029.864,A -85,B 0,C 180,E1 24340.74,E2 24340.74} C_VEL
LIN {X 0,Y 102.983,Z 1040.637,A -85,B 0,C 180,E1 24359.032,E2 24359.032} C_VEL
LIN {X 0,Y 99.891,Z 1045.041,A -85,B 0,C 180,E1 24372.354,E2 24372.354} C_VEL
LIN {X 0,Y 100.746,Z 1047.613,A -85,B 0,C 180,E1 24389.999,E2 24389.999} C_VEL
LIN {X 0,Y 99.873,Z 1045.058,A -85,B 0,C 180,E1 24407.648,E2 24407.648} C_VEL
LIN {X 0,Y 106.354,Z 1037.471,A -85,B 0,C 180,E1 24427.729,E2 24427.729} C_VEL
LIN {X 0,Y 126.332,Z 1022.557,A -85,B 0,C 180,E1 24447.023,E2 24447.023} C_VEL
LIN {X 0,Y 154.332,Z 1001.973,A -85,B 0,C 180,E1 24459.698,E2 24459.698} C_VEL
LIN {X 0,Y 185.842,Z 975.293,A -85,B 0,C 180,E1 24467.847,E2 24467.847} C_VEL
LIN {X 0,Y 215.232,Z 945.022,A -85,B 0,C 180,E1 24472.809,E2 24472.809} C_VEL
LIN {X 0,Y 224.262,Z 934.067,A -85,B 0,C 180,E1 24474.178,E2 24474.178} C_VEL
LIN {X 0,Y 225.032,Z 927.559,A -85,B 0,C 180,E1 24479.99,E2 24479.99} C_VEL
LIN {X 0,Y 225.128,Z 925.116,A -85,B 0,C 180,E1 24483.846,E2 24483.846} C_VEL
LIN {X 0,Y 222.072,Z 927.195,A -85,B 0,C 180,E1 24489.802,E2 24489.802} C_VEL
LIN {X 0,Y 218.084,Z 932.646,A -85,B 0,C 180,E1 24496.11,E2 24496.11} C_VEL
LIN {X 0,Y 216,Z 935.896,A -85,B 0,C 180,E1 24498.578,E2 24498.578} C_VEL
LIN {X 0,Y 188.608,Z 961.502,A -85,B 0,C 180,E1 24504.039,E2 24504.039} C_VEL
LIN {X 0,Y 160.229,Z 982.296,A -85,B 0,C 180,E1 24511.746,E2 24511.746} C_VEL
LIN {X 0,Y 136.131,Z 996.526,A -85,B 0,C 180,E1 24521.832,E2 24521.832} C_VEL
LIN {X 0,Y 114.729,Z 1007.002,A -85,B 0,C 180,E1 24538.14,E2 24538.14} C_VEL
LIN {X 0,Y 103.272,Z 1012.064,A -85,B 0,C 180,E1 24561.571,E2 24561.571} C_VEL
LIN {X 0,Y 103.289,Z 1012.038,A -85,B 0,C 180,E1 24578.429,E2 24578.429} C_VEL
LIN {X 0,Y 114.782,Z 1006.92,A -85,B 0,C 180,E1 24601.844,E2 24601.844} C_VEL
LIN {X 0,Y 133.659,Z 997.718,A -85,B 0,C 180,E1 24616.692,E2 24616.692} C_VEL
LIN {X 0,Y 141.213,Z 992.986,A -85,B 0,C 180,E1 24622.996,E2 24622.996} C_VEL
LIN {X 0,Y 150.039,Z 987.388,A -85,B 0,C 180,E1 24628.543,E2 24628.543} C_VEL
LIN {X 0,Y 179.239,Z 967.666,A -85,B 0,C 180,E1 24636.721,E2 24636.721} C_VEL
LIN {X 0,Y 206.89,Z 943.879,A -85,B 0,C 180,E1 24642.05,E2 24642.05} C_VEL
LIN {X 0,Y 209.903,Z 940.886,A -85,B 0,C 180,E1 24642.516,E2 24642.516} C_VEL
LIN {X 0,Y 212.95,Z 937.285,A -85,B 0,C 180,E1 24644.867,E2 24644.867} C_VEL
LIN {X 0,Y 215.844,Z 933.613,A -85,B 0,C 180,E1 24649.114,E2 24649.114} C_VEL
LIN {X 0,Y 219.66,Z 930.925,A -85,B 0,C 180,E1 24656.058,E2 24656.058} C_VEL
LIN {X 0,Y 219.401,Z 935.16,A -85,B 0,C 180,E1 24661.987,E2 24661.987} C_VEL
LIN {X 0,Y 219.026,Z 937.48,A -85,B 0,C 180,E1 24663.974,E2 24663.974} C_VEL
LIN {X 0,Y 216.556,Z 940.721,A -85,B 0,C 180,E1 24664.702,E2 24664.702} C_VEL
LIN {X 0,Y 187.898,Z 970.257,A -85,B 0,C 180,E1 24668.931,E2 24668.931} C_VEL
LIN {X 0,Y 157.258,Z 996.053,A -85,B 0,C 180,E1 24675.688,E2 24675.688} C_VEL
LIN {X 0,Y 129.941,Z 1015.628,A -85,B 0,C 180,E1 24685.447,E2 24685.447} C_VEL
LIN {X 0,Y 107.207,Z 1030.837,A -85,B 0,C 180,E1 24700.596,E2 24700.596} C_VEL
LIN {X 0,Y 94.215,Z 1040.876,A -85,B 0,C 180,E1 24721.177,E2 24721.177} C_VEL
LIN {X 0,Y 91.908,Z 1045.577,A -85,B 0,C 180,E1 24741.388,E2 24741.388} C_VEL
LIN {X 0,Y 92.882,Z 1046.25,A -85,B 0,C 180,E1 24749.999,E2 24749.999} C_VEL
LIN {X 0,Y 92.171,Z 1043.652,A -85,B 0,C 180,E1 24769.178,E2 24769.178} C_VEL
LIN {X 0,Y 99.911,Z 1036.002,A -85,B 0,C 180,E1 24790.712,E2 24790.712} C_VEL
LIN {X 0,Y 121.932,Z 1021.089,A -85,B 0,C 180,E1 24810.361,E2 24810.361} C_VEL
LIN {X 0,Y 151.699,Z 1000.383,A -85,B 0,C 180,E1 24822.755,E2 24822.755} C_VEL
LIN {X 0,Y 182.508,Z 975.364,A -85,B 0,C 180,E1 24830.091,E2 24830.091} C_VEL
LIN {X 0,Y 212.825,Z 945.17,A -85,B 0,C 180,E1 24834.825,E2 24834.825} C_VEL
LIN {X 0,Y 217.998,Z 939.351,A -85,B 0,C 180,E1 24835.46,E2 24835.46} C_VEL
LIN {X 0,Y 219.139,Z 937.61,A -85,B 0,C 180,E1 24836.028,E2 24836.028} C_VEL
LIN {X 0,Y 219.89,Z 931.975,A -85,B 0,C 180,E1 24841.962,E2 24841.962} C_VEL
LIN {X 0,Y 219.761,Z 931.098,A -85,B 0,C 180,E1 24843.94,E2 24843.94} C_VEL
LIN {X 0,Y 215.876,Z 933.858,A -85,B 0,C 180,E1 24850.933,E2 24850.933} C_VEL
LIN {X 0,Y 211.65,Z 939.207,A -85,B 0,C 180,E1 24856.614,E2 24856.614} C_VEL
LIN {X 0,Y 208.343,Z 942.67,A -85,B 0,C 180,E1 24857.656,E2 24857.656} C_VEL
LIN {X 0,Y 179.169,Z 967.904,A -85,B 0,C 180,E1 24863.228,E2 24863.228} C_VEL
LIN {X 0,Y 150.483,Z 987.261,A -85,B 0,C 180,E1 24871.222,E2 24871.222} C_VEL
LIN {X 0,Y 124.322,Z 1001.222,A -85,B 0,C 180,E1 24883.057,E2 24883.057} C_VEL
LIN {X 0,Y 104.474,Z 1009.905,A -85,B 0,C 180,E1 24900.347,E2 24900.347} C_VEL
LIN {X 0,Y 95.582,Z 1013.412,A -85,B 0,C 180,E1 24920.887,E2 24920.887} C_VEL
LIN {X 0,Y 95.599,Z 1013.386,A -85,B 0,C 180,E1 24939.113,E2 24939.113} C_VEL
LIN {X 0,Y 108.226,Z 1008.275,A -85,B 0,C 180,E1 24964.027,E2 24964.027} C_VEL
LIN {X 0,Y 131.702,Z 997.473,A -85,B 0,C 180,E1 24980.957,E2 24980.957} C_VEL
LIN {X 0,Y 150.039,Z 987.388,A -85,B 0,C 180,E1 24988.543,E2 24988.543} C_VEL
LIN {X 0,Y 159.727,Z 980.998,A -85,B 0,C 180,E1 24993.415,E2 24993.415} C_VEL
LIN {X 0,Y 169.929,Z 973.601,A -85,B 0,C 180,E1 24997.651,E2 24997.651} C_VEL
LIN {X 0,Y 197.85,Z 951.508,A -85,B 0,C 180,E1 25003.044,E2 25003.044} C_VEL
LIN {X 0,Y 205.772,Z 944.209,A -85,B 0,C 180,E1 25004.276,E2 25004.276} C_VEL
LIN {X 0,Y 210.007,Z 939.628,A -85,B 0,C 180,E1 25008.807,E2 25008.807} C_VEL
LIN {X 0,Y 214.14,Z 936.786,A -85,B 0,C 180,E1 25015.957,E2 25015.957} C_VEL
LIN {X 0,Y 213.745,Z 941.064,A -85,B 0,C 180,E1 25022.042,E2 25022.042} C_VEL
LIN {X 0,Y 212.237,Z 943.351,A -85,B 0,C 180,E1 25022.928,E2 25022.928} C_VEL
LIN {X 0,Y 183.044,Z 972.068,A -85,B 0,C 180,E1 25027,E2 25027} C_VEL
LIN {X 0,Y 151.732,Z 997.074,A -85,B 0,C 180,E1 25033.547,E2 25033.547} C_VEL
LIN {X 0,Y 120.78,Z 1017.788,A -85,B 0,C 180,E1 25044.66,E2 25044.66} C_VEL
LIN {X 0,Y 96.152,Z 1032.946,A -85,B 0,C 180,E1 25062.899,E2 25062.899} C_VEL
LIN {X 0,Y 86.089,Z 1040.421,A -85,B 0,C 180,E1 25081.607,E2 25081.607} C_VEL
LIN {X 0,Y 83.937,Z 1044.046,A -85,B 0,C 180,E1 25099.608,E2 25099.608} C_VEL
LIN {X 0,Y 85.009,Z 1044.887,A -85,B 0,C 180,E1 25109.999,E2 25109.999} C_VEL
LIN {X 0,Y 84.538,Z 1042.244,A -85,B 0,C 180,E1 25130.988,E2 25130.988} C_VEL
LIN {X 0,Y 93.733,Z 1034.555,A -85,B 0,C 180,E1 25154.046,E2 25154.046} C_VEL
LIN {X 0,Y 117.97,Z 1019.619,A -85,B 0,C 180,E1 25173.941,E2 25173.941} C_VEL
LIN {X 0,Y 150.08,Z 998.402,A -85,B 0,C 180,E1 25186.03,E2 25186.03} C_VEL
LIN {X 0,Y 181.252,Z 973.847,A -85,B 0,C 180,E1 25192.706,E2 25192.706} C_VEL
LIN {X 0,Y 212.236,Z 943.599,A -85,B 0,C 180,E1 25197.065,E2 25197.065} C_VEL
LIN {X 0,Y 213.687,Z 941.97,A -85,B 0,C 180,E1 25197.254,E2 25197.254} C_VEL
LIN {X 0,Y 214.404,Z 937.789,A -85,B 0,C 180,E1 25202.013,E2 25202.013} C_VEL
LIN {X 0,Y 214.216,Z 936.967,A -85,B 0,C 180,E1 25204.042,E2 25204.042} C_VEL
LIN {X 0,Y 209.99,Z 939.908,A -85,B 0,C 180,E1 25211.244,E2 25211.244} C_VEL
LIN {X 0,Y 206.048,Z 944.18,A -85,B 0,C 180,E1 25215.612,E2 25215.612} C_VEL
LIN {X 0,Y 176.239,Z 969.297,A -85,B 0,C 180,E1 25220.899,E2 25220.899} C_VEL
LIN {X 0,Y 146.585,Z 988.624,A -85,B 0,C 180,E1 25228.609,E2 25228.609} C_VEL
LIN {X 0,Y 119.116,Z 1002.576,A -85,B 0,C 180,E1 25240.306,E2 25240.306} C_VEL
LIN {X 0,Y 97.774,Z 1011.253,A -85,B 0,C 180,E1 25258.086,E2 25258.086} C_VEL
LIN {X 0,Y 87.888,Z 1014.763,A -85,B 0,C 180,E1 25280.081,E2 25280.081} C_VEL
LIN {X 0,Y 87.905,Z 1014.738,A -85,B 0,C 180,E1 25299.918,E2 25299.918} C_VEL
LIN {X 0,Y 101.846,Z 1009.63,A -85,B 0,C 180,E1 25326.486,E2 25326.486} C_VEL
LIN {X 0,Y 126.327,Z 999.106,A -85,B 0,C 180,E1 25343.414,E2 25343.414} C_VEL
LIN {X 0,Y 156.901,Z 982.295,A -85,B 0,C 180,E1 25354.382,E2 25354.382} C_VEL
LIN {X 0,Y 169.929,Z 973.601,A -85,B 0,C 180,E1 25357.651,E2 25357.651} C_VEL
LIN {X 0,Y 180.593,Z 965.496,A -85,B 0,C 180,E1 25361.357,E2 25361.357} C_VEL
LIN {X 0,Y 189.965,Z 957.844,A -85,B 0,C 180,E1 25364.295,E2 25364.295} C_VEL
LIN {X 0,Y 191.521,Z 956.574,A -85,B 0,C 180,E1 25364.562,E2 25364.562} C_VEL
LIN {X 0,Y 200.92,Z 948.35,A -85,B 0,C 180,E1 25365.991,E2 25365.991} C_VEL
LIN {X 0,Y 203.597,Z 945.697,A -85,B 0,C 180,E1 25368.241,E2 25368.241} C_VEL
LIN {X 0,Y 206.564,Z 943.4,A -85,B 0,C 180,E1 25372.918,E2 25372.918} C_VEL
LIN {X 0,Y 208.485,Z 942.538,A -85,B 0,C 180,E1 25375.847,E2 25375.847} C_VEL
LIN {X 0,Y 208.279,Z 945.502,A -85,B 0,C 180,E1 25380.646,E2 25380.646} C_VEL
LIN {X 0,Y 205.968,Z 948.142,A -85,B 0,C 180,E1 25381.296,E2 25381.296} C_VEL
LIN {X 0,Y 174.701,Z 976.863,A -85,B 0,C 180,E1 25385.523,E2 25385.523} C_VEL
LIN {X 0,Y 142.291,Z 1000.794,A -85,B 0,C 180,E1 25392.302,E2 25392.302} C_VEL
LIN {X 0,Y 110.431,Z 1020.35,A -85,B 0,C 180,E1 25404.306,E2 25404.306} C_VEL
LIN {X 0,Y 85.745,Z 1034.328,A -85,B 0,C 180,E1 25425.066,E2 25425.066} C_VEL
LIN {X 0,Y 76.963,Z 1040.806,A -85,B 0,C 180,E1 25446.831,E2 25446.831} C_VEL
LIN {X 0,Y 77.124,Z 1043.521,A -85,B 0,C 180,E1 25469.999,E2 25469.999} C_VEL
LIN {X 0,Y 76.963,Z 1040.829,A -85,B 0,C 180,E1 25493.167,E2 25493.167} C_VEL
LIN {X 0,Y 89.403,Z 1032.28,A -85,B 0,C 180,E1 25519.637,E2 25519.637} C_VEL
LIN {X 0,Y 117.485,Z 1016.396,A -85,B 0,C 180,E1 25539.111,E2 25539.111} C_VEL
LIN {X 0,Y 150.569,Z 995.316,A -85,B 0,C 180,E1 25549.701,E2 25549.701} C_VEL
LIN {X 0,Y 182.203,Z 970.722,A -85,B 0,C 180,E1 25555.647,E2 25555.647} C_VEL
LIN {X 0,Y 207.492,Z 946.844,A -85,B 0,C 180,E1 25558.85,E2 25558.85} C_VEL
